C03657=1186.504,380.175,-80.249,-176.015,8.629,148.561
C03658=1186.500,380.423,-80.284,-176.014,8.633,148.561
C03659=1186.496,380.670,-80.319,-176.013,8.636,148.562
C03660=1186.492,380.918,-80.354,-176.012,8.640,148.562
C03661=1186.488,381.166,-80.388,-176.011,8.643,148.563
C03662=1186.484,381.413,-80.424,-176.010,8.646,148.564
C03663=1186.479,381.661,-80.458,-176.009,8.649,148.564
C03664=1186.476,381.908,-80.494,-176.008,8.652,148.565
C03665=1186.472,382.156,-80.528,-176.007,8.655,148.565
C03666=1186.468,382.403,-80.563,-176.006,8.658,148.566
C03667=1186.464,382.651,-80.598,-176.006,8.661,148.566
C03668=1186.460,382.898,-80.632,-176.005,8.664,148.567
C03669=1186.456,383.146,-80.668,-176.004,8.667,148.567
C03670=1186.452,383.394,-80.703,-176.003,8.671,148.568
C03671=1186.448,383.641,-80.738,-176.002,8.674,148.569
C03672=1186.444,383.889,-80.773,-176.002,8.676,148.569
C03673=1186.439,384.136,-80.808,-176.001,8.680,148.570
C03674=1186.436,384.384,-80.843,-176.000,8.683,148.570
C03675=1186.432,384.631,-80.878,-175.999,8.686,148.571
C03676=1186.428,384.878,-80.912,-175.998,8.689,148.572
C03677=1186.424,385.126,-80.948,-175.998,8.692,148.572
C03678=1186.421,385.373,-80.983,-175.997,8.695,148.573
C03679=1186.416,385.621,-81.018,-175.996,8.698,148.573
C03680=1186.412,385.868,-81.053,-175.995,8.701,148.574
C03681=1186.408,386.116,-81.088,-175.994,8.704,148.574
C03682=1186.404,386.363,-81.123,-175.995,8.707,148.575
C03683=1186.400,386.611,-81.158,-175.994,8.710,148.576
C03684=1186.396,386.858,-81.193,-175.993,8.713,148.576
C03685=1186.392,387.106,-81.229,-175.992,8.716,148.577
C03686=1186.388,387.354,-81.264,-175.991,8.719,148.577
C03687=1186.384,387.600,-81.299,-175.991,8.722,148.578
C03688=1186.380,387.848,-81.335,-175.990,8.725,148.579
C03689=1186.376,388.096,-81.369,-175.990,8.728,148.579
C03690=1186.372,388.343,-81.405,-175.990,8.730,148.580
C03691=1186.368,388.591,-81.439,-175.989,8.733,148.580
C03692=1186.365,388.839,-81.475,-175.988,8.736,148.581
C03693=1186.360,389.085,-81.510,-175.988,8.739,148.582
C03694=1186.356,389.333,-81.545,-175.987,8.742,148.582
C03695=1186.353,389.581,-81.580,-175.987,8.745,148.583
C03696=1186.348,389.828,-81.616,-175.986,8.747,148.583
C03697=1186.344,390.076,-81.651,-175.985,8.751,148.584
C03698=1186.341,390.323,-81.686,-175.986,8.753,148.585
C03699=1186.337,390.570,-81.721,-175.985,8.756,148.585
C03700=1186.333,390.818,-81.757,-175.984,8.759,148.586
C03701=1186.329,391.066,-81.792,-175.984,8.762,148.587
C03702=1186.325,391.313,-81.827,-175.983,8.765,148.587
C03703=1186.321,391.560,-81.862,-175.983,8.767,148.588
C03704=1186.316,391.844,-81.902,-175.983,8.771,148.589
C03705=1186.312,392.127,-81.943,-175.982,8.774,148.589
C03706=1186.307,392.411,-81.983,-175.982,8.777,148.590
C03707=1186.303,392.695,-82.024,-175.982,8.780,148.591
C03708=1186.298,392.943,-82.060,-175.981,8.783,148.591
C03709=1186.294,393.191,-82.095,-175.981,8.785,148.592
C03710=1186.290,393.438,-82.130,-175.980,8.788,148.593
C03711=1186.286,393.685,-82.166,-175.980,8.791,148.593
C03712=1186.283,393.933,-82.201,-175.980,8.793,148.594
C03713=1186.279,394.181,-82.236,-175.980,8.796,148.594
C03714=1186.274,394.427,-82.271,-175.979,8.799,148.595
C03715=1186.271,394.675,-82.307,-175.979,8.801,148.595
C03716=1186.267,394.922,-82.342,-175.979,8.804,148.596
C03717=1186.263,395.169,-82.378,-175.978,8.807,148.597
C03718=1186.259,395.417,-82.412,-175.978,8.809,148.597
C03719=1186.255,395.665,-82.449,-175.978,8.812,148.598
C03720=1186.251,395.913,-82.484,-175.978,8.815,148.599
C03721=1186.247,396.160,-82.519,-175.977,8.817,148.599
C03722=1186.243,396.407,-82.555,-175.977,8.819,148.600
C03723=1186.239,396.655,-82.590,-175.977,8.822,148.600
C03724=1186.235,396.902,-82.625,-175.976,8.825,148.601
C03725=1186.231,397.149,-82.660,-175.977,8.827,148.602
C03726=1186.227,397.397,-82.697,-175.976,8.830,148.602
C03727=1186.223,397.645,-82.732,-175.975,8.833,148.603
C03728=1186.219,397.892,-82.767,-175.976,8.835,148.604
C03729=1186.215,398.139,-82.803,-175.975,8.838,148.604
C03730=1186.211,398.387,-82.838,-175.975,8.840,148.605
C03731=1186.208,398.634,-82.874,-175.975,8.842,148.605
C03732=1186.203,398.881,-82.908,-175.975,8.845,148.606
C03733=1186.199,399.129,-82.945,-175.975,8.847,148.607
C03734=1186.195,399.377,-82.980,-175.974,8.850,148.607
C03735=1186.191,399.624,-83.016,-175.974,8.853,148.608
C03736=1186.187,399.871,-83.051,-175.974,8.855,148.608
C03737=1186.184,400.119,-83.086,-175.974,8.857,148.609
C03738=1186.179,400.366,-83.122,-175.974,8.860,148.609
C03739=1186.175,400.614,-83.158,-175.974,8.862,148.610
C03740=1186.171,400.861,-83.193,-175.974,8.864,148.611
C03741=1186.168,401.108,-83.229,-175.974,8.867,148.611
C03742=1186.164,401.356,-83.264,-175.974,8.869,148.612
C03743=1186.160,401.603,-83.300,-175.974,8.872,148.612
C03744=1186.156,401.851,-83.336,-175.973,8.874,148.613
C03745=1186.152,402.098,-83.371,-175.973,8.876,148.614
C03746=1186.148,402.346,-83.406,-175.973,8.879,148.614
C03747=1186.144,402.593,-83.442,-175.973,8.881,148.615
C03748=1186.140,402.841,-83.477,-175.973,8.883,148.615
C03749=1186.135,403.088,-83.513,-175.973,8.886,148.616
C03750=1186.132,403.336,-83.548,-175.973,8.888,148.616
C03751=1186.128,403.583,-83.584,-175.973,8.891,148.617
C03752=1186.124,403.831,-83.620,-175.973,8.893,148.618
C03753=1186.120,404.078,-83.656,-175.972,8.895,148.618
C03754=1186.116,404.325,-83.691,-175.972,8.897,148.619
C03755=1186.112,404.573,-83.726,-175.973,8.899,148.619
C03756=1186.108,404.820,-83.762,-175.973,8.901,148.620
C03757=1186.105,405.068,-83.798,-175.972,8.904,148.620
C03758=1186.100,405.315,-83.833,-175.972,8.906,148.621
C03759=1186.096,405.562,-83.869,-175.972,8.908,148.622
C03760=1186.092,405.810,-83.904,-175.972,8.911,148.622
C03761=1186.089,406.057,-83.940,-175.972,8.913,148.623
C03762=1186.085,406.304,-83.977,-175.972,8.916,148.623
C03763=1186.080,406.551,-84.012,-175.972,8.917,148.624
C03764=1186.077,406.799,-84.048,-175.972,8.919,148.624
C03765=1186.073,407.046,-84.083,-175.972,8.922,148.625
C03766=1186.069,407.294,-84.119,-175.972,8.924,148.626
C03767=1186.065,407.542,-84.155,-175.972,8.926,148.626
C03768=1186.061,407.789,-84.190,-175.972,8.928,148.627
C03769=1186.057,408.036,-84.225,-175.972,8.930,148.627
C03770=1186.053,408.284,-84.262,-175.972,8.933,148.628
C03771=1186.049,408.531,-84.297,-175.972,8.935,148.628
C03772=1186.045,408.779,-84.333,-175.971,8.937,148.629
C03773=1186.041,409.026,-84.369,-175.972,8.939,148.629
C03774=1186.037,409.273,-84.404,-175.972,8.941,148.630
C03775=1186.033,409.521,-84.440,-175.972,8.943,148.631
C03776=1186.029,409.768,-84.475,-175.971,8.946,148.631
C03777=1186.025,410.015,-84.512,-175.972,8.947,148.632
C03778=1186.021,410.263,-84.548,-175.971,8.949,148.632
C03779=1186.018,410.510,-84.583,-175.971,8.952,148.633
C03780=1186.014,410.757,-84.618,-175.971,8.954,148.633
C03781=1186.009,411.005,-84.654,-175.972,8.956,148.634
C03782=1186.005,411.253,-84.690,-175.971,8.958,148.634
C03783=1186.002,411.500,-84.726,-175.971,8.960,148.635
C03784=1185.997,411.748,-84.762,-175.971,8.962,148.635
C03785=1185.993,411.995,-84.797,-175.971,8.964,148.636
C03786=1185.990,412.242,-84.833,-175.971,8.966,148.637
C03787=1185.985,412.489,-84.869,-175.972,8.968,148.637
C03788=1185.982,412.737,-84.905,-175.971,8.970,148.638
C03789=1185.978,412.984,-84.940,-175.971,8.972,148.638
C03790=1185.974,413.232,-84.976,-175.971,8.974,148.639
C03791=1185.970,413.480,-85.012,-175.971,8.976,148.639
C03792=1185.966,413.726,-85.047,-175.971,8.978,148.640
C03793=1185.962,413.973,-85.083,-175.972,8.980,148.640
C03794=1185.958,414.221,-85.120,-175.971,8.982,148.641
C03795=1185.954,414.469,-85.155,-175.971,8.985,148.641
C03796=1185.951,414.716,-85.191,-175.971,8.986,148.642
C03797=1185.946,414.964,-85.227,-175.971,8.988,148.642
C03798=1185.942,415.211,-85.262,-175.971,8.990,148.643
C03799=1185.939,415.458,-85.298,-175.971,8.992,148.643
C03800=1185.932,415.876,-85.359,-175.971,8.996,148.644
C03801=1185.928,416.294,-85.419,-175.971,8.998,148.645
C03802=1185.928,416.711,-85.479,-175.971,9.002,148.646
C03803=1185.931,417.128,-85.538,-175.971,9.005,148.647
C03804=1185.510,417.129,-85.580,-175.974,9.016,148.650
C03805=1185.507,416.919,-85.550,-175.974,9.014,148.650
C03806=1185.506,416.709,-85.520,-175.974,9.012,148.649
C03807=1185.506,416.499,-85.490,-175.974,9.011,148.649
C03808=1185.506,416.289,-85.460,-175.974,9.009,148.649
C03809=1185.508,416.078,-85.429,-175.974,9.008,148.648
C03810=1185.510,415.868,-85.399,-175.974,9.006,148.648
C03811=1185.513,415.657,-85.368,-175.974,9.004,148.647
C03812=1185.517,415.448,-85.338,-175.974,9.003,148.647
C03813=1185.521,415.200,-85.302,-175.974,9.001,148.647
C03814=1185.525,414.952,-85.266,-175.974,8.999,148.646
C03815=1185.529,414.705,-85.231,-175.974,8.997,148.645
C03816=1185.533,414.457,-85.195,-175.974,8.995,148.645
C03817=1185.537,414.210,-85.158,-175.974,8.993,148.644
C03818=1185.540,413.963,-85.123,-175.975,8.991,148.644
C03819=1185.545,413.716,-85.088,-175.974,8.989,148.644
C03820=1185.549,413.468,-85.051,-175.975,8.987,148.643
C03821=1185.553,413.221,-85.016,-175.974,8.985,148.642
C03822=1185.556,412.973,-84.980,-175.974,8.983,148.642
C03823=1185.560,412.726,-84.944,-175.974,8.981,148.641
C03824=1185.564,412.478,-84.908,-175.974,8.979,148.641
C03825=1185.568,412.232,-84.873,-175.974,8.977,148.640
C03826=1185.573,411.984,-84.837,-175.975,8.975,148.640
C03827=1185.576,411.736,-84.801,-175.974,8.973,148.639
C03828=1185.580,411.489,-84.766,-175.974,8.971,148.639
C03829=1185.584,411.241,-84.730,-175.974,8.969,148.638
C03830=1185.588,410.993,-84.694,-175.975,8.966,148.638
C03831=1185.592,410.747,-84.658,-175.974,8.965,148.637
C03832=1185.596,410.500,-84.622,-175.975,8.963,148.637
C03833=1185.600,410.252,-84.586,-175.974,8.960,148.636
C03834=1185.604,410.004,-84.551,-175.974,8.959,148.635
C03835=1185.608,409.757,-84.515,-175.974,8.956,148.635
C03836=1185.611,409.509,-84.480,-175.975,8.954,148.634
C03837=1185.616,409.262,-84.444,-175.975,8.952,148.634
C03838=1185.620,409.015,-84.408,-175.974,8.950,148.633
C03839=1185.623,408.767,-84.373,-175.974,8.948,148.633
C03840=1185.628,408.520,-84.336,-175.975,8.946,148.632
C03841=1185.631,408.273,-84.300,-175.975,8.943,148.632
C03842=1185.635,408.025,-84.265,-175.974,8.942,148.631
C03843=1185.639,407.778,-84.230,-175.974,8.939,148.630
C03844=1185.644,407.531,-84.193,-175.975,8.937,148.630
C03845=1185.647,407.283,-84.158,-175.975,8.935,148.629
C03846=1185.651,407.036,-84.122,-175.975,8.932,148.629
C03847=1185.655,406.788,-84.087,-175.974,8.931,148.628
C03848=1185.660,406.541,-84.051,-175.975,8.929,148.628
C03849=1185.663,406.293,-84.016,-175.975,8.926,148.627
C03850=1185.667,406.046,-83.980,-175.975,8.924,148.626
C03851=1185.671,405.798,-83.944,-175.975,8.921,148.626
C03852=1185.675,405.551,-83.908,-175.975,8.919,148.625
C03853=1185.679,405.304,-83.873,-175.974,8.917,148.625
C03854=1185.683,405.056,-83.838,-175.975,8.915,148.624
C03855=1185.687,404.809,-83.802,-175.975,8.913,148.624
C03856=1185.691,404.561,-83.766,-175.975,8.911,148.623
C03857=1185.695,404.314,-83.730,-175.975,8.908,148.622
C03858=1185.699,404.067,-83.695,-175.975,8.906,148.622
C03859=1185.703,403.819,-83.660,-175.976,8.904,148.621
C03860=1185.707,403.571,-83.623,-175.975,8.901,148.621
C03861=1185.711,403.324,-83.588,-175.976,8.899,148.620
C03862=1185.714,403.076,-83.552,-175.976,8.896,148.620
C03863=1185.719,402.830,-83.517,-175.976,8.894,148.619
C03864=1185.722,402.582,-83.482,-175.976,8.892,148.618
C03865=1185.727,402.334,-83.445,-175.976,8.889,148.618
C03866=1185.730,402.087,-83.410,-175.976,8.887,148.617
C03867=1185.735,401.840,-83.375,-175.976,8.885,148.617
C03868=1185.738,401.593,-83.339,-175.976,8.883,148.616
C03869=1185.743,401.345,-83.303,-175.976,8.880,148.615
C03870=1185.746,401.097,-83.268,-175.977,8.877,148.615
C03871=1185.750,400.850,-83.232,-175.977,8.875,148.614
C03872=1185.754,400.603,-83.197,-175.977,8.873,148.614
C03873=1185.758,400.355,-83.161,-175.977,8.870,148.613
C03874=1185.761,400.108,-83.126,-175.977,8.868,148.612
C03875=1185.766,399.860,-83.090,-175.977,8.865,148.612
C03876=1185.770,399.613,-83.054,-175.977,8.863,148.611
C03877=1185.774,399.366,-83.019,-175.977,8.861,148.611
C03878=1185.777,399.118,-82.983,-175.977,8.858,148.610
C03879=1185.781,398.871,-82.948,-175.978,8.856,148.610
C03880=1185.786,398.623,-82.913,-175.977,8.854,148.609
C03881=1185.790,398.376,-82.877,-175.978,8.851,148.608
C03882=1185.794,398.128,-82.842,-175.979,8.848,148.608
C03883=1185.797,397.881,-82.806,-175.978,8.846,148.607
C03884=1185.802,397.634,-82.771,-175.979,8.843,148.606
C03885=1185.805,397.386,-82.735,-175.978,8.841,148.606
C03886=1185.809,397.139,-82.700,-175.979,8.839,148.605
C03887=1185.813,396.891,-82.664,-175.979,8.836,148.605
C03888=1185.818,396.644,-82.629,-175.979,8.833,148.604
C03889=1185.822,396.396,-82.594,-175.980,8.831,148.603
C03890=1185.825,396.149,-82.558,-175.980,8.828,148.603
C03891=1185.830,395.902,-82.523,-175.980,8.826,148.602
C03892=1185.833,395.654,-82.487,-175.980,8.823,148.602
C03893=1185.837,395.407,-82.452,-175.981,8.820,148.601
C03894=1185.841,395.159,-82.416,-175.980,8.818,148.600
C03895=1185.846,394.912,-82.381,-175.981,8.815,148.600
C03896=1185.850,394.664,-82.346,-175.981,8.812,148.599
C03897=1185.853,394.417,-82.310,-175.981,8.810,148.598
C03898=1185.857,394.169,-82.275,-175.982,8.807,148.598
C03899=1185.861,393.922,-82.239,-175.982,8.804,148.597
C03900=1185.865,393.674,-82.204,-175.982,8.802,148.597
C03901=1185.869,393.427,-82.169,-175.983,8.799,148.596
C03902=1185.873,393.180,-82.134,-175.983,8.796,148.595
C03903=1185.877,392.932,-82.098,-175.983,8.794,148.595
C03904=1185.881,392.684,-82.062,-175.984,8.791,148.594
C03905=1185.886,392.400,-82.022,-175.984,8.788,148.593
C03906=1185.890,392.117,-81.981,-175.985,8.784,148.593
C03907=1185.895,391.833,-81.941,-175.985,8.782,148.592
C03908=1185.899,391.550,-81.900,-175.985,8.778,148.591
C03909=1185.903,391.302,-81.866,-175.986,8.775,148.591
C03910=1185.907,391.054,-81.830,-175.986,8.773,148.590
C03911=1185.911,390.807,-81.795,-175.987,8.770,148.589
C03912=1185.915,390.560,-81.759,-175.987,8.767,148.589
C03913=1185.919,390.312,-81.724,-175.988,8.764,148.588
C03914=1185.923,390.065,-81.689,-175.988,8.762,148.588
C03915=1185.927,389.817,-81.654,-175.988,8.759,148.587
C03916=1185.931,389.569,-81.619,-175.989,8.756,148.586
C03917=1185.935,389.322,-81.584,-175.989,8.753,148.586
C03918=1185.939,389.075,-81.548,-175.990,8.750,148.585
C03919=1185.943,388.827,-81.513,-175.991,8.747,148.585
C03920=1185.947,388.580,-81.478,-175.991,8.745,148.584
C03921=1185.951,388.333,-81.443,-175.992,8.741,148.583
C03922=1185.955,388.084,-81.408,-175.992,8.738,148.583
C03923=1185.959,387.838,-81.373,-175.992,8.736,148.582
C03924=1185.963,387.590,-81.337,-175.993,8.733,148.582
C03925=1185.966,387.342,-81.302,-175.994,8.730,148.581
C03926=1185.971,387.095,-81.267,-175.994,8.727,148.580
C03927=1185.974,386.848,-81.231,-175.995,8.724,148.580
C03928=1185.978,386.600,-81.197,-175.995,8.721,148.579
C03929=1185.983,386.353,-81.161,-175.996,8.718,148.578
C03930=1185.987,386.105,-81.127,-175.997,8.715,148.578
C03931=1185.990,385.857,-81.091,-175.998,8.712,148.577
C03932=1185.995,385.610,-81.056,-175.998,8.709,148.577
C03933=1185.999,385.362,-81.021,-175.999,8.706,148.576
C03934=1186.003,385.115,-80.986,-176.000,8.703,148.576
C03935=1186.007,384.867,-80.951,-176.001,8.700,148.575
C03936=1186.010,384.620,-80.915,-176.001,8.697,148.574
C03937=1186.015,384.372,-80.881,-176.002,8.694,148.574
C03938=1186.019,384.125,-80.845,-176.002,8.690,148.573
C03939=1186.023,383.877,-80.811,-176.003,8.687,148.573
C03940=1186.027,383.630,-80.775,-176.004,8.684,148.572
C03941=1186.030,383.382,-80.741,-176.005,8.681,148.571
C03942=1186.034,383.135,-80.706,-176.006,8.678,148.571
C03943=1186.038,382.887,-80.671,-176.007,8.675,148.570
C03944=1186.042,382.640,-80.636,-176.008,8.672,148.570
C03945=1186.047,382.392,-80.601,-176.009,8.669,148.569
C03946=1186.050,382.145,-80.566,-176.009,8.666,148.569
C03947=1186.055,381.897,-80.531,-176.010,8.663,148.568
C03948=1186.058,381.650,-80.496,-176.011,8.660,148.567
C03949=1186.062,381.402,-80.461,-176.012,8.657,148.567
C03950=1186.066,381.155,-80.426,-176.013,8.653,148.566
C03951=1186.070,380.907,-80.391,-176.014,8.650,148.566
C03952=1186.074,380.660,-80.357,-176.015,8.647,148.565
C03953=1186.078,380.412,-80.321,-176.016,8.644,148.565
C03954=1186.083,380.165,-80.287,-176.017,8.641,148.564
C03955=1186.086,379.917,-80.251,-176.018,8.638,148.564
C03956=1186.090,379.669,-80.217,-176.019,8.634,148.563
C03957=1186.094,379.422,-80.183,-176.020,8.631,148.562
C03958=1186.098,379.175,-80.147,-176.021,8.628,148.562
C03959=1186.102,378.927,-80.113,-176.022,8.625,148.561
C03960=1186.106,378.679,-80.078,-176.023,8.621,148.561
C03961=1186.111,378.432,-80.043,-176.024,8.618,148.560
C03962=1186.115,378.184,-80.008,-176.025,8.615,148.560
C03963=1186.118,377.937,-79.974,-176.027,8.611,148.559
C03964=1186.122,377.690,-79.938,-176.028,8.608,148.559
C03965=1186.127,377.442,-79.904,-176.029,8.605,148.558
C03966=1186.131,377.194,-79.869,-176.030,8.601,148.557
C03967=1186.135,376.947,-79.835,-176.031,8.598,148.557
C03968=1186.138,376.699,-79.800,-176.032,8.595,148.557
C03969=1186.143,376.452,-79.765,-176.034,8.591,148.556
C03970=1186.147,376.204,-79.730,-176.035,8.588,148.556
C03971=1186.151,375.956,-79.696,-176.036,8.585,148.555
C03972=1186.154,375.709,-79.661,-176.037,8.581,148.554
C03973=1186.158,375.461,-79.626,-176.038,8.579,148.554
C03974=1186.163,375.214,-79.592,-176.040,8.575,148.553
C03975=1186.166,374.966,-79.557,-176.041,8.572,148.553
C03976=1186.170,374.719,-79.522,-176.042,8.568,148.552
C03977=1186.174,374.471,-79.487,-176.043,8.565,148.552
C03978=1186.179,374.224,-79.453,-176.045,8.561,148.551
C03979=1186.183,373.976,-79.419,-176.046,8.559,148.551
C03980=1186.187,373.728,-79.384,-176.047,8.555,148.550
C03981=1186.191,373.481,-79.350,-176.049,8.552,148.550
C03982=1186.194,373.233,-79.316,-176.051,8.548,148.549
C03983=1186.199,372.986,-79.280,-176.051,8.545,148.549
C03984=1186.203,372.738,-79.245,-176.053,8.541,148.548
C03985=1186.206,372.491,-79.212,-176.054,8.539,148.548
C03986=1186.210,372.243,-79.177,-176.056,8.535,148.547
C03987=1186.215,371.996,-79.142,-176.057,8.532,148.547
C03988=1186.218,371.748,-79.108,-176.059,8.528,148.547
C03989=1186.223,371.500,-79.074,-176.060,8.524,148.546
C03990=1186.227,371.252,-79.039,-176.061,8.522,148.546
C03991=1186.231,371.005,-79.005,-176.063,8.518,148.545
C03992=1186.235,370.758,-78.970,-176.064,8.515,148.544
C03993=1186.238,370.510,-78.936,-176.066,8.511,148.544
C03994=1186.243,370.262,-78.902,-176.068,8.508,148.544
C03995=1186.247,370.014,-78.867,-176.069,8.505,148.543
C03996=1186.251,369.767,-78.833,-176.071,8.501,148.543
C03997=1186.255,369.519,-78.798,-176.072,8.497,148.542
C03998=1186.259,369.272,-78.764,-176.073,8.494,148.542
C03999=1186.263,369.025,-78.730,-176.075,8.491,148.541
C04000=1186.267,368.776,-78.695,-176.077,8.487,148.541
C04001=1186.271,368.529,-78.661,-176.078,8.484,148.541
C04002=1186.275,368.282,-78.627,-176.080,8.481,148.540
C04003=1186.279,368.034,-78.592,-176.082,8.477,148.540
C04004=1186.284,367.786,-78.559,-176.083,8.474,148.539
C04005=1186.287,367.538,-78.524,-176.085,8.471,148.539
C04006=1186.291,367.291,-78.490,-176.087,8.467,148.538
C04007=1186.295,367.044,-78.456,-176.088,8.463,148.538
C04008=1186.299,366.796,-78.421,-176.089,8.460,148.537
C04009=1186.304,366.515,-78.383,-176.092,8.456,148.537
C04010=1186.308,366.234,-78.344,-176.093,8.452,148.536
C04011=1186.313,365.951,-78.305,-176.095,8.449,148.536
C04012=1186.317,365.670,-78.266,-176.097,8.445,148.536
C04013=1186.321,365.423,-78.232,-176.099,8.441,148.535
C04014=1186.326,365.176,-78.198,-176.101,8.438,148.535
C04015=1186.329,364.928,-78.164,-176.102,8.434,148.534
C04016=1186.334,364.680,-78.130,-176.105,8.431,148.534
C04017=1186.338,364.433,-78.096,-176.106,8.428,148.534
C04018=1186.342,364.184,-78.061,-176.108,8.424,148.533
C04019=1186.346,363.937,-78.028,-176.110,8.421,148.533
C04020=1186.350,363.690,-77.994,-176.111,8.417,148.532
C04021=1186.354,363.441,-77.959,-176.113,8.414,148.532
C04022=1186.357,363.194,-77.926,-176.115,8.410,148.532
C04023=1186.362,362.946,-77.892,-176.117,8.407,148.531
C04024=1186.366,362.699,-77.858,-176.119,8.404,148.531
C04025=1186.370,362.451,-77.824,-176.120,8.400,148.530
C04026=1186.374,362.203,-77.790,-176.123,8.397,148.530
C04027=1186.378,361.956,-77.756,-176.124,8.393,148.530
C04028=1186.382,361.708,-77.723,-176.126,8.390,148.529
C04029=1186.386,361.460,-77.688,-176.128,8.386,148.529
C04030=1186.390,361.213,-77.655,-176.130,8.384,148.529
C04031=1186.394,360.965,-77.621,-176.131,8.380,148.528
C04032=1186.398,360.717,-77.586,-176.134,8.377,148.528
C04033=1186.402,360.470,-77.553,-176.136,8.373,148.528
C04034=1186.406,360.223,-77.519,-176.138,8.370,148.527
C04035=1186.410,359.974,-77.485,-176.140,8.366,148.527
C04036=1186.414,359.727,-77.451,-176.141,8.362,148.527
C04037=1186.418,359.479,-77.418,-176.144,8.359,148.526
C04038=1186.422,359.232,-77.384,-176.145,8.355,148.526
C04039=1186.426,358.983,-77.350,-176.148,8.352,148.526
C04040=1186.430,358.736,-77.316,-176.150,8.349,148.525
C04041=1186.434,358.488,-77.283,-176.151,8.346,148.525
C04042=1186.438,358.241,-77.249,-176.153,8.342,148.525
C04043=1186.443,357.993,-77.215,-176.155,8.339,148.524
C04044=1186.447,357.745,-77.182,-176.157,8.335,148.524
C04045=1186.451,357.498,-77.148,-176.159,8.332,148.524
C04046=1186.455,357.250,-77.115,-176.162,8.329,148.524
C04047=1186.460,357.002,-77.081,-176.163,8.325,148.523
C04048=1186.463,356.755,-77.047,-176.166,8.322,148.523
C04049=1186.467,356.506,-77.014,-176.167,8.318,148.522
C04050=1186.471,356.259,-76.980,-176.170,8.315,148.522
C04051=1186.475,356.012,-76.947,-176.172,8.312,148.522
C04052=1186.479,355.764,-76.914,-176.174,8.308,148.522
C04053=1186.484,355.516,-76.880,-176.176,8.305,148.521
C04054=1186.488,355.269,-76.846,-176.178,8.301,148.521
C04055=1186.491,355.020,-76.812,-176.180,8.298,148.521
C04056=1186.495,354.772,-76.779,-176.182,8.294,148.521
C04057=1186.500,354.525,-76.746,-176.185,8.291,148.520
C04058=1186.503,354.278,-76.712,-176.186,8.287,148.520
C04059=1186.508,354.030,-76.679,-176.189,8.284,148.520
C04060=1186.512,353.782,-76.645,-176.191,8.281,148.519
C04061=1186.517,353.534,-76.612,-176.193,8.277,148.519
C04062=1186.520,353.286,-76.578,-176.195,8.274,148.519
C04063=1186.524,353.039,-76.545,-176.197,8.271,148.519
C04064=1186.528,352.791,-76.512,-176.199,8.268,148.518
C04065=1186.532,352.543,-76.478,-176.201,8.264,148.518
C04066=1186.536,352.295,-76.445,-176.203,8.261,148.518
C04067=1186.540,352.048,-76.412,-176.205,8.258,148.517
C04068=1186.545,351.800,-76.379,-176.207,8.254,148.517
C04069=1186.549,351.552,-76.346,-176.210,8.251,148.517
C04070=1186.553,351.305,-76.313,-176.211,8.248,148.517
C04071=1186.557,351.057,-76.279,-176.214,8.244,148.516
C04072=1186.561,350.810,-76.246,-176.216,8.241,148.516
C04073=1186.565,350.562,-76.213,-176.218,8.238,148.516
C04074=1186.569,350.314,-76.179,-176.220,8.234,148.516
C04075=1186.573,350.066,-76.146,-176.223,8.231,148.515
C04076=1186.577,349.818,-76.113,-176.225,8.227,148.515
C04077=1186.581,349.570,-76.080,-176.227,8.224,148.515
C04078=1186.585,349.323,-76.046,-176.229,8.221,148.515
C04079=1186.589,349.075,-76.013,-176.231,8.217,148.514
C04080=1186.593,348.827,-75.980,-176.234,8.214,148.514
C04081=1186.597,348.579,-75.947,-176.235,8.212,148.514
C04082=1186.602,348.331,-75.914,-176.237,8.208,148.514
C04083=1186.606,348.083,-75.881,-176.240,8.205,148.514
C04084=1186.610,347.836,-75.848,-176.242,8.202,148.513
C04085=1186.614,347.588,-75.815,-176.244,8.198,148.513
C04086=1186.618,347.340,-75.782,-176.246,8.195,148.513
C04087=1186.623,347.092,-75.749,-176.248,8.191,148.512
C04088=1186.627,346.845,-75.716,-176.251,8.188,148.512
C04089=1186.630,346.597,-75.683,-176.253,8.185,148.512
C04090=1186.635,346.349,-75.651,-176.255,8.181,148.512
C04091=1186.639,346.101,-75.617,-176.257,8.178,148.512
C04092=1186.643,345.853,-75.584,-176.260,8.175,148.511
C04093=1186.647,345.606,-75.551,-176.262,8.171,148.511
C04094=1186.651,345.358,-75.518,-176.264,8.168,148.511
C04095=1186.656,345.110,-75.485,-176.266,8.165,148.511
C04096=1186.659,344.862,-75.453,-176.269,8.161,148.511
C04097=1186.663,344.614,-75.420,-176.270,8.159,148.510
C04098=1186.668,344.367,-75.387,-176.272,8.156,148.510
C04099=1186.672,344.119,-75.355,-176.275,8.152,148.510
C04100=1186.676,343.871,-75.321,-176.277,8.149,148.510
C04101=1186.680,343.624,-75.289,-176.280,8.146,148.510
C04102=1186.684,343.376,-75.256,-176.282,8.143,148.509
C04103=1186.688,343.128,-75.223,-176.284,8.139,148.509
C04104=1186.693,342.880,-75.190,-176.286,8.136,148.509
C04105=1186.697,342.632,-75.158,-176.289,8.133,148.509
C04106=1186.700,342.384,-75.125,-176.291,8.129,148.509
C04107=1186.705,342.136,-75.093,-176.293,8.126,148.508
C04108=1186.709,341.888,-75.059,-176.295,8.123,148.508
C04109=1186.714,341.641,-75.027,-176.298,8.119,148.508
C04110=1186.717,341.393,-74.995,-176.300,8.116,148.508
C04111=1186.722,341.146,-74.962,-176.303,8.113,148.508
C04112=1186.726,340.897,-74.929,-176.304,8.111,148.508
C04113=1186.730,340.619,-74.893,-176.307,8.106,148.507
C04114=1186.735,340.340,-74.856,-176.309,8.103,148.507
C04115=1186.740,340.061,-74.819,-176.312,8.099,148.507
C04116=1186.745,339.783,-74.782,-176.314,8.096,148.507
C04117=1186.748,339.535,-74.751,-176.317,8.093,148.507
C04118=1186.753,339.286,-74.718,-176.319,8.089,148.506
C04119=1186.757,339.039,-74.685,-176.322,8.086,148.506
C04120=1186.761,338.790,-74.653,-176.324,8.083,148.506
C04121=1186.765,338.543,-74.620,-176.326,8.079,148.506
C04122=1186.770,338.295,-74.588,-176.329,8.076,148.506
C04123=1186.773,338.048,-74.555,-176.331,8.073,148.505
C04124=1186.778,337.799,-74.523,-176.333,8.071,148.505
C04125=1186.781,337.551,-74.491,-176.335,8.067,148.505
C04126=1186.785,337.304,-74.458,-176.337,8.064,148.505
C04127=1186.789,337.056,-74.426,-176.340,8.061,148.505
C04128=1186.794,336.808,-74.394,-176.342,8.058,148.505
C04129=1186.798,336.560,-74.361,-176.345,8.054,148.504
C04130=1186.802,336.312,-74.329,-176.347,8.051,148.504
C04131=1186.807,336.064,-74.296,-176.350,8.048,148.504
C04132=1186.810,335.816,-74.264,-176.352,8.045,148.504
C04133=1186.815,335.569,-74.232,-176.354,8.041,148.504
C04134=1186.819,335.321,-74.200,-176.357,8.038,148.504
C04135=1186.823,335.072,-74.168,-176.359,8.035,148.504
C04136=1186.826,334.825,-74.135,-176.361,8.032,148.503
C04137=1186.832,334.577,-74.103,-176.363,8.029,148.503
C04138=1186.835,334.329,-74.071,-176.366,8.026,148.503
C04139=1186.840,334.081,-74.039,-176.368,8.023,148.503
C04140=1186.843,333.833,-74.007,-176.370,8.019,148.503
C04141=1186.848,333.586,-73.974,-176.373,8.016,148.503
C04142=1186.852,333.338,-73.942,-176.375,8.013,148.503
C04143=1186.856,333.090,-73.910,-176.377,8.010,148.502
C04144=1186.860,332.841,-73.878,-176.380,8.007,148.502
C04145=1186.864,332.594,-73.846,-176.382,8.003,148.502
C04146=1186.869,332.346,-73.814,-176.384,8.001,148.502
C04147=1186.872,332.098,-73.782,-176.387,7.998,148.502
C04148=1186.877,331.850,-73.750,-176.389,7.995,148.502
C04149=1186.881,331.602,-73.718,-176.392,7.992,148.502
C04150=1186.885,331.354,-73.686,-176.394,7.988,148.502
C04151=1186.890,331.107,-73.654,-176.396,7.985,148.501
C04152=1186.893,330.859,-73.622,-176.399,7.982,148.501
C04153=1186.897,330.611,-73.590,-176.401,7.979,148.501
C04154=1186.902,330.363,-73.558,-176.403,7.975,148.501
C04155=1186.906,330.115,-73.526,-176.406,7.972,148.501
C04156=1186.910,329.867,-73.494,-176.408,7.969,148.501
C04157=1186.915,329.619,-73.463,-176.410,7.967,148.501
C04158=1186.919,329.371,-73.431,-176.413,7.964,148.501
C04159=1186.922,329.123,-73.399,-176.415,7.960,148.500
C04160=1186.927,328.875,-73.367,-176.418,7.957,148.500
C04161=1186.931,328.627,-73.335,-176.420,7.954,148.500
C04162=1186.935,328.379,-73.303,-176.423,7.951,148.500
C04163=1186.940,328.131,-73.271,-176.425,7.948,148.500
C04164=1186.943,327.883,-73.239,-176.428,7.945,148.500
C04165=1186.947,327.635,-73.208,-176.430,7.941,148.500
C04166=1186.952,327.388,-73.176,-176.432,7.939,148.500
C04167=1186.956,327.139,-73.144,-176.434,7.936,148.500
C04168=1186.961,326.892,-73.113,-176.437,7.933,148.500
C04169=1186.964,326.644,-73.081,-176.439,7.929,148.499
C04170=1186.968,326.396,-73.049,-176.441,7.926,148.499
C04171=1186.972,326.148,-73.018,-176.444,7.923,148.499
C04172=1186.977,325.899,-72.986,-176.446,7.920,148.499
C04173=1186.981,325.652,-72.954,-176.449,7.917,148.499
C04174=1186.985,325.404,-72.923,-176.451,7.913,148.499
C04175=1186.989,325.157,-72.891,-176.453,7.911,148.499
C04176=1186.993,324.908,-72.860,-176.456,7.908,148.499
C04177=1186.998,324.659,-72.828,-176.458,7.905,148.499
C04178=1187.002,324.412,-72.796,-176.461,7.902,148.498
C04179=1187.006,324.163,-72.765,-176.463,7.899,148.498
C04180=1187.010,323.916,-72.733,-176.466,7.896,148.498
C04181=1187.014,323.668,-72.702,-176.468,7.892,148.498
C04182=1187.019,323.420,-72.671,-176.471,7.889,148.498
C04183=1187.022,323.172,-72.639,-176.473,7.887,148.498
C04184=1187.027,322.925,-72.608,-176.475,7.884,148.498
C04185=1187.031,322.676,-72.576,-176.478,7.880,148.498
C04186=1187.034,322.428,-72.545,-176.480,7.877,148.498
C04187=1187.040,322.180,-72.513,-176.483,7.874,148.498
C04188=1187.044,321.932,-72.481,-176.485,7.871,148.498
C04189=1187.048,321.684,-72.451,-176.488,7.868,148.497
C04190=1187.052,321.436,-72.419,-176.490,7.865,148.497
C04191=1187.056,321.188,-72.388,-176.492,7.863,148.497
C04192=1187.060,320.940,-72.356,-176.495,7.859,148.497
C04193=1187.065,320.692,-72.325,-176.497,7.856,148.497
C04194=1187.069,320.444,-72.294,-176.500,7.853,148.497
C04195=1187.073,320.196,-72.263,-176.502,7.850,148.497
C04196=1187.077,319.949,-72.231,-176.505,7.847,148.497
C04197=1187.081,319.700,-72.200,-176.507,7.844,148.497
C04198=1187.086,319.453,-72.169,-176.510,7.841,148.497
C04199=1187.090,319.204,-72.138,-176.512,7.838,148.497
C04200=1187.094,318.957,-72.106,-176.514,7.835,148.497
C04201=1187.098,318.708,-72.075,-176.517,7.832,148.497
C04202=1187.103,318.460,-72.044,-176.519,7.829,148.497
C04203=1187.106,318.212,-72.012,-176.522,7.826,148.497
C04204=1187.111,317.964,-71.982,-176.524,7.822,148.496
C04205=1187.115,317.716,-71.951,-176.527,7.819,148.496
C04206=1187.119,317.468,-71.920,-176.529,7.817,148.496
C04207=1187.123,317.220,-71.889,-176.531,7.814,148.496
C04208=1187.127,316.972,-71.858,-176.534,7.811,148.496
C04209=1187.132,316.724,-71.826,-176.537,7.808,148.496
C04210=1187.136,316.476,-71.795,-176.539,7.805,148.496
C04211=1187.140,316.228,-71.764,-176.542,7.802,148.496
C04212=1187.145,315.980,-71.734,-176.545,7.799,148.496
C04213=1187.148,315.732,-71.702,-176.546,7.796,148.496
C04214=1187.152,315.484,-71.672,-176.549,7.793,148.496
C04215=1187.157,315.236,-71.641,-176.552,7.790,148.496
C04216=1187.161,314.987,-71.610,-176.554,7.787,148.496
C04217=1187.166,314.712,-71.575,-176.557,7.784,148.496
C04218=1187.171,314.435,-71.540,-176.560,7.780,148.496
C04219=1187.175,314.158,-71.506,-176.563,7.777,148.496
C04220=1187.180,313.882,-71.472,-176.565,7.774,148.496
C04221=1187.184,313.633,-71.441,-176.568,7.771,148.496
C04222=1187.189,313.385,-71.410,-176.570,7.768,148.496
C04223=1187.193,313.137,-71.379,-176.573,7.764,148.495
C04224=1187.196,312.889,-71.349,-176.575,7.762,148.495
C04225=1187.201,312.642,-71.317,-176.577,7.759,148.495
C04226=1187.205,312.394,-71.286,-176.580,7.756,148.495
C04227=1187.209,312.145,-71.255,-176.582,7.753,148.495
C04228=1187.213,311.897,-71.225,-176.585,7.750,148.495
C04229=1187.218,311.649,-71.194,-176.588,7.747,148.495
C04230=1187.222,311.401,-71.163,-176.589,7.744,148.495
C04231=1187.226,311.153,-71.133,-176.592,7.741,148.495
C04232=1187.230,310.905,-71.102,-176.595,7.738,148.495
C04233=1187.235,310.657,-71.072,-176.598,7.735,148.495
C04234=1187.239,310.408,-71.040,-176.600,7.732,148.495
C04235=1187.243,310.161,-71.010,-176.603,7.729,148.495
C04236=1187.248,309.912,-70.980,-176.605,7.727,148.495
C04237=1187.252,309.664,-70.949,-176.607,7.724,148.495
C04238=1187.256,309.416,-70.919,-176.610,7.720,148.495
C04239=1187.260,309.168,-70.888,-176.612,7.717,148.495
C04240=1187.265,308.920,-70.857,-176.615,7.714,148.495
C04241=1187.269,308.672,-70.827,-176.618,7.711,148.495
C04242=1187.273,308.424,-70.796,-176.619,7.709,148.495
C04243=1187.277,308.176,-70.765,-176.622,7.706,148.495
C04244=1187.282,307.928,-70.736,-176.625,7.703,148.495
C04245=1187.286,307.680,-70.705,-176.628,7.700,148.495
C04246=1187.289,307.431,-70.675,-176.630,7.697,148.495
C04247=1187.294,307.183,-70.644,-176.633,7.694,148.495
C04248=1187.299,306.935,-70.613,-176.635,7.691,148.495
C04249=1187.303,306.687,-70.584,-176.637,7.688,148.495
C04250=1187.307,306.439,-70.553,-176.640,7.685,148.495
C04251=1187.311,306.191,-70.523,-176.642,7.682,148.494
C04252=1187.315,305.943,-70.492,-176.645,7.679,148.494
C04253=1187.320,305.694,-70.462,-176.647,7.677,148.495
C04254=1187.324,305.447,-70.431,-176.650,7.674,148.495
C04255=1187.328,305.199,-70.401,-176.653,7.671,148.495
C04256=1187.333,304.950,-70.371,-176.655,7.668,148.494
C04257=1187.337,304.703,-70.341,-176.658,7.665,148.494
C04258=1187.341,304.454,-70.310,-176.660,7.662,148.494
C04259=1187.345,304.206,-70.280,-176.663,7.659,148.494
C04260=1187.350,303.958,-70.250,-176.665,7.656,148.495
C04261=1187.354,303.710,-70.219,-176.668,7.653,148.495
C04262=1187.358,303.462,-70.189,-176.670,7.650,148.494
C04263=1187.362,303.214,-70.159,-176.672,7.648,148.494
C04264=1187.367,302.965,-70.129,-176.675,7.645,148.494
C04265=1187.371,302.717,-70.099,-176.678,7.642,148.494
C04266=1187.375,302.468,-70.069,-176.680,7.639,148.494
C04267=1187.379,302.221,-70.038,-176.683,7.636,148.494
C04268=1187.383,301.972,-70.009,-176.685,7.633,148.494
C04269=1187.388,301.725,-69.978,-176.688,7.630,148.494
C04270=1187.392,301.476,-69.949,-176.690,7.627,148.494
C04271=1187.397,301.228,-69.918,-176.693,7.624,148.494
C04272=1187.401,300.980,-69.889,-176.696,7.621,148.494
C04273=1187.405,300.732,-69.858,-176.698,7.619,148.494
C04274=1187.410,300.484,-69.828,-176.701,7.616,148.494
C04275=1187.414,300.236,-69.798,-176.703,7.613,148.494
C04276=1187.418,299.988,-69.769,-176.706,7.610,148.494
C04277=1187.422,299.739,-69.738,-176.708,7.607,148.494
C04278=1187.426,299.491,-69.708,-176.710,7.605,148.494
C04279=1187.430,299.243,-69.679,-176.713,7.602,148.494
C04280=1187.435,298.995,-69.648,-176.716,7.599,148.494
C04281=1187.439,298.746,-69.618,-176.719,7.596,148.494
C04282=1187.443,298.498,-69.589,-176.721,7.594,148.495
C04283=1187.448,298.250,-69.558,-176.723,7.591,148.495
C04284=1187.452,298.002,-69.529,-176.726,7.587,148.494
C04285=1187.456,297.754,-69.499,-176.728,7.584,148.494
C04286=1187.460,297.506,-69.469,-176.731,7.581,148.494
C04287=1187.465,297.257,-69.439,-176.733,7.579,148.494
C04288=1187.469,297.009,-69.410,-176.736,7.576,148.495
C04289=1187.473,296.761,-69.380,-176.739,7.573,148.495
C04290=1187.477,296.513,-69.350,-176.741,7.570,148.495
C04291=1187.482,296.265,-69.320,-176.744,7.568,148.495
C04292=1187.486,296.016,-69.291,-176.746,7.565,148.495
C04293=1187.491,295.768,-69.261,-176.749,7.562,148.495
C04294=1187.495,295.520,-69.232,-176.752,7.559,148.495
C04295=1187.499,295.272,-69.201,-176.753,7.557,148.495
C04296=1187.503,295.024,-69.172,-176.756,7.554,148.495
C04297=1187.508,294.775,-69.142,-176.759,7.551,148.495
C04298=1187.512,294.527,-69.112,-176.762,7.548,148.495
C04299=1187.516,294.279,-69.083,-176.764,7.545,148.495
C04300=1187.520,294.031,-69.054,-176.766,7.542,148.495
C04301=1187.524,293.782,-69.024,-176.769,7.539,148.495
C04302=1187.529,293.534,-68.995,-176.772,7.536,148.495
C04303=1187.533,293.287,-68.965,-176.774,7.534,148.495
C04304=1187.538,293.039,-68.935,-176.777,7.531,148.495
C04305=1187.542,292.790,-68.905,-176.779,7.528,148.495
C04306=1187.546,292.542,-68.876,-176.782,7.525,148.495
C04307=1187.551,292.294,-68.846,-176.784,7.523,148.495
C04308=1187.555,292.045,-68.817,-176.787,7.520,148.495
C04309=1187.559,291.797,-68.788,-176.790,7.517,148.495
C04310=1187.563,291.549,-68.758,-176.792,7.514,148.495
C04311=1187.567,291.301,-68.729,-176.795,7.512,148.495
C04312=1187.571,291.052,-68.699,-176.797,7.509,148.495
C04313=1187.576,290.804,-68.670,-176.800,7.506,148.495
C04314=1187.580,290.557,-68.641,-176.802,7.503,148.495
C04315=1187.585,290.308,-68.612,-176.804,7.500,148.495
C04316=1187.589,290.059,-68.582,-176.807,7.497,148.495
C04317=1187.593,289.811,-68.553,-176.810,7.494,148.495
C04318=1187.597,289.563,-68.524,-176.813,7.491,148.495
C04319=1187.602,289.315,-68.494,-176.815,7.489,148.495
C04320=1187.606,289.066,-68.465,-176.817,7.486,148.495
C04321=1187.611,288.792,-68.432,-176.820,7.483,148.495
C04322=1187.616,288.518,-68.400,-176.823,7.481,148.496
C04323=1187.621,288.243,-68.367,-176.826,7.478,148.496
C04324=1187.626,287.968,-68.336,-176.829,7.475,148.496
C04325=1187.630,287.720,-68.306,-176.831,7.472,148.496
C04326=1187.634,287.472,-68.277,-176.834,7.469,148.496
C04327=1187.638,287.223,-68.247,-176.837,7.466,148.496
C04328=1187.643,286.975,-68.219,-176.839,7.463,148.496
C04329=1187.647,286.727,-68.190,-176.842,7.460,148.496
C04330=1187.651,286.479,-68.161,-176.845,7.457,148.496
C04331=1187.655,286.231,-68.131,-176.847,7.455,148.496
C04332=1187.660,285.982,-68.103,-176.849,7.452,148.496
C04333=1187.664,285.734,-68.073,-176.852,7.449,148.496
C04334=1187.669,285.486,-68.044,-176.855,7.446,148.496
C04335=1187.673,285.237,-68.015,-176.857,7.444,148.496
C04336=1187.677,284.989,-67.986,-176.860,7.441,148.496
C04337=1187.681,284.742,-67.957,-176.862,7.438,148.496
C04338=1187.686,284.493,-67.929,-176.865,7.436,148.496
C04339=1187.690,284.244,-67.899,-176.867,7.433,148.496
C04340=1187.694,283.996,-67.870,-176.870,7.430,148.496
C04341=1187.699,283.748,-67.841,-176.873,7.427,148.496
C04342=1187.703,283.500,-67.812,-176.875,7.425,148.496
C04343=1187.707,283.251,-67.784,-176.878,7.422,148.496
C04344=1187.711,283.003,-67.754,-176.880,7.419,148.496
C04345=1187.716,282.755,-67.726,-176.882,7.417,148.497
C04346=1187.721,282.506,-67.696,-176.885,7.414,148.497
C04347=1187.724,282.258,-67.668,-176.888,7.411,148.497
C04348=1187.729,282.010,-67.639,-176.891,7.409,148.497
C04349=1187.734,281.761,-67.610,-176.893,7.406,148.497
C04350=1187.738,281.513,-67.581,-176.896,7.403,148.497
C04351=1187.742,281.265,-67.553,-176.898,7.401,148.497
C04352=1187.747,281.016,-67.525,-176.901,7.398,148.497
C04353=1187.751,280.768,-67.495,-176.904,7.395,148.497
C04354=1187.755,280.519,-67.466,-176.906,7.392,148.497
C04355=1187.759,280.272,-67.438,-176.908,7.389,148.497
C04356=1187.764,280.023,-67.409,-176.911,7.386,148.497
C04357=1187.768,279.775,-67.380,-176.913,7.384,148.497
C04358=1187.772,279.527,-67.352,-176.916,7.381,148.497
C04359=1187.777,279.278,-67.323,-176.919,7.378,148.497
C04360=1187.780,279.030,-67.294,-176.921,7.376,148.497
C04361=1187.785,278.782,-67.266,-176.924,7.373,148.498
C04362=1187.790,278.533,-67.237,-176.927,7.370,148.498
C04363=1187.794,278.286,-67.209,-176.929,7.368,148.498
C04364=1187.798,278.037,-67.180,-176.932,7.365,148.498
C04365=1187.803,277.788,-67.151,-176.934,7.362,148.498
C04366=1187.807,277.540,-67.123,-176.937,7.360,148.498
C04367=1187.811,277.292,-67.094,-176.939,7.357,148.498
C04368=1187.815,277.043,-67.066,-176.942,7.354,148.498
C04369=1187.820,276.795,-67.037,-176.944,7.352,148.498
C04370=1187.824,276.546,-67.009,-176.947,7.349,148.498
C04371=1187.829,276.299,-66.980,-176.950,7.346,148.498
C04372=1187.833,276.050,-66.951,-176.952,7.344,148.499
C04373=1187.837,275.801,-66.923,-176.955,7.341,148.499
C04374=1187.842,275.553,-66.895,-176.958,7.338,148.499
C04375=1187.846,275.305,-66.867,-176.960,7.336,148.499
C04376=1187.851,275.057,-66.838,-176.963,7.333,148.499
C04377=1187.854,274.809,-66.810,-176.965,7.330,148.499
C04378=1187.859,274.560,-66.781,-176.968,7.328,148.499
C04379=1187.863,274.312,-66.753,-176.971,7.325,148.499
C04380=1187.868,274.063,-66.724,-176.973,7.323,148.499
C04381=1187.872,273.815,-66.697,-176.975,7.320,148.499
C04382=1187.877,273.566,-66.668,-176.978,7.317,148.499
C04383=1187.881,273.318,-66.640,-176.980,7.315,148.499
C04384=1187.885,273.070,-66.612,-176.983,7.312,148.499
C04385=1187.890,272.822,-66.584,-176.986,7.309,148.500
C04386=1187.893,272.573,-66.555,-176.988,7.307,148.500
C04387=1187.899,272.325,-66.527,-176.991,7.304,148.500
C04388=1187.902,272.076,-66.499,-176.993,7.302,148.500
C04389=1187.907,271.828,-66.470,-176.996,7.299,148.500
C04390=1187.911,271.579,-66.442,-176.999,7.296,148.500
C04391=1187.916,271.332,-66.415,-177.001,7.294,148.500
C04392=1187.920,271.083,-66.386,-177.004,7.291,148.500
C04393=1187.924,270.835,-66.358,-177.007,7.288,148.500
C04394=1187.929,270.586,-66.329,-177.009,7.286,148.500
C04395=1187.933,270.338,-66.302,-177.012,7.283,148.500
C04396=1187.937,270.089,-66.273,-177.014,7.281,148.501
C04397=1187.942,269.841,-66.246,-177.017,7.278,148.501
C04398=1187.947,269.593,-66.218,-177.020,7.275,148.501
C04399=1187.950,269.344,-66.190,-177.022,7.273,148.501
C04400=1187.956,269.096,-66.161,-177.025,7.270,148.501
C04401=1187.959,268.847,-66.133,-177.027,7.268,148.501
C04402=1187.964,268.600,-66.106,-177.030,7.265,148.501
C04403=1187.968,268.350,-66.078,-177.033,7.262,148.501
C04404=1187.973,268.102,-66.050,-177.035,7.260,148.501
C04405=1187.977,267.854,-66.022,-177.038,7.257,148.501
C04406=1187.981,267.606,-65.994,-177.040,7.255,148.502
C04407=1187.986,267.357,-65.966,-177.042,7.252,148.502
C04408=1187.990,267.108,-65.938,-177.046,7.249,148.502
C04409=1187.994,266.860,-65.910,-177.048,7.247,148.502
C04410=1187.998,266.612,-65.882,-177.051,7.244,148.502
C04411=1188.004,266.363,-65.854,-177.053,7.242,148.502
C04412=1188.008,266.115,-65.827,-177.055,7.239,148.502
C04413=1188.012,265.867,-65.799,-177.059,7.236,148.502
C04414=1188.016,265.618,-65.771,-177.061,7.234,148.502
C04415=1188.021,265.370,-65.743,-177.064,7.231,148.503
C04416=1188.025,265.121,-65.715,-177.066,7.229,148.503
C04417=1188.030,264.873,-65.688,-177.069,7.226,148.503
C04418=1188.034,264.624,-65.660,-177.071,7.224,148.503
C04419=1188.038,264.376,-65.632,-177.074,7.221,148.503
C04420=1188.043,264.128,-65.605,-177.076,7.218,148.503
C04421=1188.047,263.879,-65.576,-177.079,7.216,148.503
C04422=1188.052,263.631,-65.549,-177.082,7.213,148.503
C04423=1188.056,263.383,-65.521,-177.084,7.211,148.503
C04424=1188.060,263.133,-65.494,-177.087,7.208,148.504
C04425=1188.065,262.861,-65.464,-177.090,7.205,148.504
C04426=1188.071,262.588,-65.433,-177.093,7.202,148.504
C04427=1188.075,262.315,-65.403,-177.095,7.199,148.504
C04428=1188.080,262.043,-65.373,-177.098,7.198,148.504
C04429=1188.084,261.794,-65.345,-177.101,7.195,148.504
C04430=1188.088,261.545,-65.318,-177.103,7.192,148.504
C04431=1188.093,261.298,-65.290,-177.106,7.190,148.505
C04432=1188.097,261.048,-65.262,-177.109,7.187,148.505
C04433=1188.101,260.801,-65.235,-177.111,7.185,148.505
C04434=1188.106,260.552,-65.208,-177.114,7.182,148.505
C04435=1188.110,260.304,-65.181,-177.116,7.180,148.505
C04436=1188.114,260.055,-65.152,-177.119,7.177,148.505
C04437=1188.119,259.806,-65.125,-177.121,7.175,148.505
C04438=1188.123,259.558,-65.098,-177.124,7.172,148.505
C04439=1188.128,259.310,-65.071,-177.127,7.170,148.506
C04440=1188.132,259.061,-65.043,-177.129,7.167,148.506
C04441=1188.136,258.812,-65.016,-177.131,7.165,148.506
C04442=1188.141,258.565,-64.988,-177.135,7.162,148.506
C04443=1188.145,258.316,-64.961,-177.137,7.159,148.506
C04444=1188.149,258.067,-64.934,-177.140,7.157,148.506
C04445=1188.154,257.819,-64.906,-177.142,7.154,148.506
C04446=1188.158,257.570,-64.879,-177.145,7.152,148.506
C04447=1188.163,257.322,-64.852,-177.148,7.149,148.507
C04448=1188.167,257.073,-64.824,-177.150,7.147,148.507
C04449=1188.172,256.825,-64.797,-177.153,7.144,148.507
C04450=1188.176,256.576,-64.770,-177.155,7.142,148.507
C04451=1188.181,256.328,-64.743,-177.158,7.139,148.507
C04452=1188.185,256.079,-64.715,-177.161,7.137,148.507
C04453=1188.190,255.831,-64.688,-177.163,7.134,148.507
C04454=1188.194,255.582,-64.660,-177.165,7.132,148.508
C04455=1188.198,255.334,-64.634,-177.169,7.129,148.508
C04456=1188.202,255.086,-64.607,-177.171,7.127,148.508
C04457=1188.207,254.837,-64.580,-177.173,7.124,148.508
C04458=1188.212,254.589,-64.553,-177.176,7.122,148.508
C04459=1188.216,254.340,-64.526,-177.179,7.119,148.508
C04460=1188.220,254.091,-64.498,-177.181,7.117,148.508
C04461=1188.225,253.842,-64.471,-177.184,7.115,148.509
C04462=1188.229,253.595,-64.444,-177.186,7.112,148.509
C04463=1188.233,253.346,-64.417,-177.189,7.109,148.509
C04464=1188.238,253.098,-64.390,-177.192,7.108,148.509
C04465=1188.243,252.849,-64.363,-177.194,7.105,148.509
C04466=1188.247,252.601,-64.336,-177.197,7.102,148.509
C04467=1188.251,252.352,-64.309,-177.200,7.100,148.510
C04468=1188.255,252.104,-64.282,-177.202,7.098,148.510
C04469=1188.260,251.855,-64.255,-177.205,7.095,148.510
C04470=1188.265,251.607,-64.228,-177.207,7.093,148.510
C04471=1188.269,251.358,-64.201,-177.210,7.090,148.510
C04472=1188.273,251.110,-64.174,-177.212,7.088,148.510
C04473=1188.278,250.861,-64.148,-177.215,7.085,148.510
C04474=1188.282,250.613,-64.121,-177.218,7.083,148.511
C04475=1188.287,250.364,-64.094,-177.220,7.081,148.511
C04476=1188.291,250.116,-64.067,-177.223,7.078,148.511
C04477=1188.296,249.867,-64.040,-177.225,7.076,148.511
C04478=1188.299,249.618,-64.013,-177.228,7.073,148.511
C04479=1188.304,249.370,-63.986,-177.231,7.071,148.511
C04480=1188.309,249.121,-63.959,-177.233,7.068,148.511
C04481=1188.313,248.873,-63.933,-177.236,7.066,148.512
C04482=1188.318,248.624,-63.906,-177.239,7.063,148.512
C04483=1188.322,248.375,-63.879,-177.241,7.061,148.512
C04484=1188.326,248.127,-63.853,-177.244,7.058,148.512
C04485=1188.331,247.879,-63.826,-177.246,7.056,148.512
C04486=1188.336,247.630,-63.799,-177.249,7.054,148.513
C04487=1188.340,247.381,-63.773,-177.252,7.052,148.513
C04488=1188.344,247.133,-63.746,-177.254,7.049,148.513
C04489=1188.348,246.885,-63.719,-177.257,7.047,148.513
C04490=1188.353,246.636,-63.692,-177.259,7.045,148.513
C04491=1188.358,246.387,-63.666,-177.262,7.042,148.513
C04492=1188.362,246.139,-63.640,-177.264,7.040,148.513
C04493=1188.367,245.890,-63.612,-177.268,7.037,148.514
C04494=1188.371,245.642,-63.587,-177.270,7.035,148.514
C04495=1188.375,245.393,-63.560,-177.273,7.032,148.514
C04496=1188.379,245.145,-63.533,-177.275,7.030,148.514
C04497=1188.384,244.896,-63.507,-177.277,7.028,148.514
C04498=1188.388,244.648,-63.480,-177.281,7.025,148.515
C04499=1188.393,244.399,-63.453,-177.283,7.023,148.515
C04500=1188.397,244.150,-63.428,-177.286,7.020,148.515
C04501=1188.402,243.902,-63.401,-177.288,7.018,148.515
C04502=1188.406,243.653,-63.375,-177.291,7.015,148.515
C04503=1188.411,243.405,-63.348,-177.293,7.014,148.515
C04504=1188.415,243.156,-63.322,-177.296,7.011,148.516
C04505=1188.420,242.908,-63.295,-177.299,7.009,148.516
C04506=1188.424,242.660,-63.269,-177.301,7.007,148.516
C04507=1188.429,242.411,-63.242,-177.304,7.004,148.516
C04508=1188.433,242.163,-63.216,-177.306,7.002,148.516
C04509=1188.438,241.913,-63.190,-177.309,7.000,148.517
C04510=1188.442,241.665,-63.163,-177.312,6.997,148.517
C04511=1188.447,241.416,-63.137,-177.314,6.995,148.517
C04512=1188.451,241.168,-63.110,-177.317,6.992,148.517
C04513=1188.455,240.919,-63.085,-177.319,6.990,148.517
C04514=1188.460,240.671,-63.059,-177.322,6.988,148.518
C04515=1188.464,240.423,-63.032,-177.325,6.985,148.518
C04516=1188.469,240.173,-63.006,-177.327,6.983,148.518
C04517=1188.473,239.925,-62.979,-177.330,6.980,148.518
C04518=1188.477,239.676,-62.954,-177.333,6.979,148.518
C04519=1188.482,239.427,-62.927,-177.335,6.976,148.518
C04520=1188.486,239.179,-62.901,-177.338,6.974,148.519
C04521=1188.491,238.930,-62.875,-177.340,6.972,148.519
C04522=1188.496,238.682,-62.849,-177.343,6.969,148.519
C04523=1188.500,238.434,-62.823,-177.346,6.967,148.519
C04524=1188.504,238.185,-62.797,-177.348,6.965,148.519
C04525=1188.509,237.936,-62.770,-177.351,6.962,148.520
C04526=1188.513,237.688,-62.744,-177.354,6.960,148.520
C04527=1188.517,237.439,-62.718,-177.356,6.957,148.520
C04528=1188.523,237.190,-62.692,-177.359,6.955,148.520
C04529=1188.527,236.919,-62.664,-177.362,6.952,148.520
C04530=1188.532,236.647,-62.635,-177.364,6.951,148.521
C04531=1188.536,236.376,-62.607,-177.368,6.948,148.521
C04532=1188.542,236.104,-62.578,-177.370,6.945,148.521
C04533=1188.547,235.856,-62.553,-177.373,6.943,148.521
C04534=1188.551,235.607,-62.527,-177.375,6.941,148.521
C04535=1188.555,235.359,-62.501,-177.378,6.938,148.522
C04536=1188.560,235.109,-62.474,-177.380,6.936,148.522
C04537=1188.565,234.861,-62.449,-177.383,6.934,148.522
C04538=1188.569,234.613,-62.423,-177.386,6.931,148.522
C04539=1188.573,234.364,-62.397,-177.388,6.929,148.523
C04540=1188.577,234.115,-62.372,-177.391,6.927,148.523
C04541=1188.583,233.867,-62.345,-177.394,6.925,148.523
C04542=1188.587,233.618,-62.319,-177.396,6.923,148.523
C04543=1188.591,233.370,-62.293,-177.399,6.920,148.523
C04544=1188.595,233.121,-62.268,-177.402,6.918,148.524
C04545=1188.600,232.873,-62.242,-177.404,6.916,148.524
C04546=1188.604,232.624,-62.216,-177.407,6.913,148.524
C04547=1188.609,232.375,-62.190,-177.409,6.911,148.524
C04548=1188.614,232.127,-62.165,-177.412,6.909,148.524
C04549=1188.618,231.878,-62.139,-177.415,6.906,148.525
C04550=1188.622,231.629,-62.113,-177.417,6.904,148.525
C04551=1188.627,231.380,-62.087,-177.420,6.902,148.525
C04552=1188.632,231.132,-62.062,-177.423,6.900,148.525
C04553=1188.636,230.883,-62.036,-177.425,6.898,148.526
C04554=1188.640,230.634,-62.011,-177.428,6.896,148.526
C04555=1188.645,230.386,-61.985,-177.431,6.893,148.526
C04556=1188.649,230.138,-61.959,-177.433,6.891,148.526
C04557=1188.654,229.888,-61.933,-177.436,6.889,148.526
C04558=1188.659,229.640,-61.908,-177.438,6.886,148.526
C04559=1188.663,229.392,-61.882,-177.441,6.884,148.527
C04560=1188.668,229.142,-61.857,-177.444,6.882,148.527
C04561=1188.672,228.894,-61.832,-177.446,6.880,148.527
C04562=1188.677,228.645,-61.806,-177.449,6.878,148.528
C04563=1188.681,228.396,-61.780,-177.451,6.876,148.528
C04564=1188.686,228.148,-61.755,-177.454,6.873,148.528
C04565=1188.690,227.900,-61.729,-177.457,6.871,148.528
C04566=1188.694,227.650,-61.704,-177.459,6.869,148.528
C04567=1188.699,227.402,-61.678,-177.462,6.866,148.529
C04568=1188.703,227.153,-61.653,-177.465,6.864,148.529
C04569=1188.708,226.905,-61.627,-177.467,6.862,148.529
C04570=1188.713,226.656,-61.602,-177.471,6.860,148.529
C04571=1188.717,226.407,-61.577,-177.473,6.858,148.530
C04572=1188.722,226.159,-61.551,-177.475,6.856,148.530
C04573=1188.725,225.910,-61.526,-177.478,6.854,148.530
C04574=1188.730,225.661,-61.500,-177.481,6.851,148.530
C04575=1188.735,225.413,-61.476,-177.483,6.849,148.531
C04576=1188.739,225.164,-61.450,-177.486,6.847,148.531
C04577=1188.744,224.916,-61.424,-177.489,6.844,148.531
C04578=1188.748,224.666,-61.399,-177.491,6.842,148.531
C04579=1188.753,224.418,-61.374,-177.494,6.840,148.531
C04580=1188.757,224.169,-61.348,-177.497,6.838,148.532
C04581=1188.762,223.920,-61.323,-177.499,6.836,148.532
C04582=1188.767,223.672,-61.298,-177.502,6.834,148.532
C04583=1188.770,223.423,-61.273,-177.504,6.832,148.532
C04584=1188.775,223.175,-61.248,-177.507,6.829,148.533
C04585=1188.780,222.926,-61.222,-177.510,6.827,148.533
C04586=1188.785,222.677,-61.198,-177.512,6.825,148.533
C04587=1188.789,222.428,-61.172,-177.515,6.822,148.533
C04588=1188.794,222.180,-61.147,-177.518,6.821,148.534
C04589=1188.798,221.931,-61.122,-177.520,6.819,148.534
C04590=1188.802,221.683,-61.097,-177.523,6.817,148.534
C04591=1188.807,221.434,-61.072,-177.526,6.814,148.534
C04592=1188.812,221.186,-61.046,-177.528,6.812,148.535
C04593=1188.816,220.936,-61.021,-177.531,6.810,148.535
C04594=1188.820,220.688,-60.996,-177.533,6.808,148.535
C04595=1188.825,220.439,-60.971,-177.536,6.805,148.535
C04596=1188.830,220.191,-60.946,-177.539,6.803,148.536
C04597=1188.834,219.941,-60.921,-177.541,6.802,148.536
C04598=1188.839,219.693,-60.897,-177.544,6.799,148.536
C04599=1188.843,219.444,-60.871,-177.547,6.797,148.536
C04600=1188.848,219.195,-60.846,-177.549,6.795,148.537
C04601=1188.852,218.947,-60.821,-177.552,6.793,148.537
C04602=1188.857,218.698,-60.797,-177.555,6.790,148.537
C04603=1188.861,218.449,-60.772,-177.557,6.788,148.537
C04604=1188.866,218.201,-60.746,-177.560,6.787,148.538
C04605=1188.870,217.952,-60.722,-177.562,6.784,148.538
C04606=1188.875,217.703,-60.696,-177.565,6.782,148.538
C04607=1188.880,217.455,-60.672,-177.568,6.780,148.538
C04608=1188.884,217.206,-60.647,-177.570,6.778,148.539
C04609=1188.889,216.957,-60.623,-177.573,6.776,148.539
C04610=1188.893,216.708,-60.597,-177.576,6.773,148.539
C04611=1188.897,216.460,-60.573,-177.579,6.772,148.540
C04612=1188.902,216.210,-60.548,-177.581,6.769,148.540
C04613=1188.907,215.962,-60.522,-177.584,6.768,148.540
C04614=1188.911,215.714,-60.498,-177.587,6.765,148.540
C04615=1188.916,215.464,-60.473,-177.589,6.763,148.540
C04616=1188.920,215.216,-60.449,-177.592,6.761,148.541
C04617=1188.924,214.967,-60.423,-177.594,6.759,148.541
C04618=1188.929,214.718,-60.399,-177.597,6.757,148.541
C04619=1188.934,214.470,-60.375,-177.600,6.754,148.542
C04620=1188.938,214.221,-60.350,-177.602,6.753,148.542
C04621=1188.943,213.972,-60.326,-177.605,6.751,148.542
C04622=1188.948,213.723,-60.301,-177.607,6.749,148.542
C04623=1188.951,213.475,-60.276,-177.610,6.746,148.543
C04624=1188.956,213.226,-60.251,-177.613,6.744,148.543
C04625=1188.961,212.978,-60.227,-177.616,6.742,148.543
C04626=1188.965,212.728,-60.202,-177.618,6.740,148.543
C04627=1188.970,212.480,-60.178,-177.621,6.738,148.544
C04628=1188.974,212.231,-60.153,-177.624,6.736,148.544
C04629=1188.979,211.982,-60.129,-177.626,6.734,148.544
C04630=1188.984,211.733,-60.104,-177.629,6.732,148.545
C04631=1188.988,211.485,-60.080,-177.631,6.730,148.545
C04632=1188.993,211.236,-60.055,-177.634,6.727,148.545
C04633=1188.998,210.965,-60.028,-177.637,6.726,148.546
C04634=1189.003,210.695,-60.002,-177.640,6.723,148.546
C04635=1189.008,210.424,-59.975,-177.642,6.721,148.546
C04636=1189.012,210.155,-59.948,-177.646,6.718,148.546
C04637=1189.017,209.906,-59.924,-177.648,6.716,148.547
C04638=1189.021,209.657,-59.900,-177.651,6.715,148.547
C04639=1189.026,209.408,-59.875,-177.654,6.713,148.547
C04640=1189.030,209.160,-59.851,-177.656,6.711,148.547
C04641=1189.036,208.910,-59.827,-177.659,6.708,148.548
C04642=1189.040,208.661,-59.802,-177.662,6.706,148.548
C04643=1189.044,208.413,-59.778,-177.664,6.704,148.548
C04644=1189.049,208.164,-59.753,-177.667,6.702,148.548
C04645=1189.054,207.916,-59.729,-177.669,6.700,148.549
C04646=1189.057,207.666,-59.705,-177.672,6.698,148.549
C04647=1189.062,207.418,-59.680,-177.675,6.696,148.549
C04648=1189.067,207.169,-59.656,-177.677,6.694,148.550
C04649=1189.072,206.921,-59.631,-177.680,6.692,148.550
C04650=1189.077,206.672,-59.608,-177.683,6.690,148.550
C04651=1189.080,206.422,-59.584,-177.686,6.688,148.551
C04652=1189.086,206.174,-59.559,-177.688,6.686,148.551
C04653=1189.090,205.925,-59.535,-177.691,6.684,148.551
C04654=1189.094,205.677,-59.511,-177.693,6.682,148.551
C04655=1189.100,205.428,-59.487,-177.696,6.680,148.552
C04656=1189.104,205.178,-59.462,-177.699,6.678,148.552
C04657=1189.108,204.930,-59.438,-177.701,6.675,148.552
C04658=1189.112,204.682,-59.414,-177.704,6.673,148.553
C04659=1189.118,204.432,-59.390,-177.707,6.672,148.553
C04660=1189.122,204.184,-59.366,-177.709,6.670,148.553
C04661=1189.126,203.935,-59.342,-177.712,6.668,148.554
C04662=1189.131,203.686,-59.318,-177.714,6.666,148.554
C04663=1189.136,203.437,-59.294,-177.717,6.663,148.554
C04664=1189.140,203.189,-59.270,-177.720,6.661,148.554
C04665=1189.145,202.939,-59.246,-177.723,6.660,148.555
C04666=1189.149,202.691,-59.222,-177.725,6.658,148.555
C04667=1189.153,202.442,-59.198,-177.728,6.656,148.555
C04668=1189.159,202.193,-59.174,-177.730,6.654,148.555
C04669=1189.163,201.944,-59.150,-177.733,6.651,148.556
C04670=1189.167,201.696,-59.126,-177.736,6.649,148.556
C04671=1189.172,201.447,-59.102,-177.739,6.648,148.556
C04672=1189.176,201.198,-59.078,-177.741,6.645,148.557
C04673=1189.182,200.949,-59.054,-177.744,6.644,148.557
C04674=1189.186,200.700,-59.030,-177.746,6.642,148.557
C04675=1189.190,200.451,-59.007,-177.749,6.640,148.558
C04676=1189.195,200.202,-58.982,-177.752,6.637,148.558
C04677=1189.199,199.954,-58.958,-177.755,6.636,148.558
C04678=1189.204,199.705,-58.935,-177.757,6.633,148.558
C04679=1189.208,199.457,-58.911,-177.760,6.632,148.559
C04680=1189.213,199.208,-58.888,-177.762,6.630,148.559
C04681=1189.218,198.959,-58.863,-177.765,6.628,148.559
C04682=1189.223,198.710,-58.840,-177.768,6.626,148.560
C04683=1189.228,198.461,-58.816,-177.770,6.624,148.560
C04684=1189.232,198.212,-58.792,-177.773,6.621,148.560
C04685=1189.237,197.963,-58.769,-177.776,6.620,148.561
C04686=1189.240,197.714,-58.744,-177.778,6.618,148.561
C04687=1189.245,197.465,-58.721,-177.781,6.616,148.561
C04688=1189.250,197.217,-58.697,-177.784,6.614,148.562
C04689=1189.254,196.968,-58.674,-177.786,6.612,148.562
C04690=1189.259,196.719,-58.650,-177.789,6.610,148.562
C04691=1189.263,196.470,-58.626,-177.791,6.609,148.562
C04692=1189.268,196.221,-58.603,-177.794,6.606,148.563
C04693=1189.273,195.972,-58.579,-177.797,6.604,148.563
C04694=1189.277,195.724,-58.555,-177.800,6.602,148.563
C04695=1189.282,195.475,-58.532,-177.802,6.601,148.564
C04696=1189.286,195.226,-58.509,-177.805,6.599,148.564
C04697=1189.291,194.977,-58.485,-177.807,6.597,148.564
C04698=1189.296,194.728,-58.461,-177.810,6.595,148.565
C04699=1189.300,194.479,-58.438,-177.813,6.593,148.565
C04700=1189.305,194.230,-58.414,-177.815,6.591,148.565
C04701=1189.309,193.982,-58.390,-177.818,6.589,148.566
C04702=1189.314,193.733,-58.367,-177.821,6.587,148.566
C04703=1189.319,193.484,-58.344,-177.824,6.585,148.566
C04704=1189.323,193.235,-58.320,-177.826,6.583,148.567
C04705=1189.328,192.986,-58.296,-177.829,6.581,148.567
C04706=1189.333,192.737,-58.273,-177.831,6.579,148.567
C04707=1189.337,192.488,-58.250,-177.834,6.577,148.568
C04708=1189.341,192.240,-58.227,-177.837,6.576,148.568
C04709=1189.347,191.991,-58.204,-177.839,6.574,148.568
C04710=1189.351,191.742,-58.180,-177.842,6.572,148.569
C04711=1189.356,191.494,-58.156,-177.845,6.570,148.569
C04712=1189.360,191.245,-58.133,-177.847,6.568,148.569
C04713=1189.365,190.996,-58.110,-177.849,6.566,148.569
C04714=1189.370,190.747,-58.086,-177.853,6.564,148.570
C04715=1189.374,190.498,-58.063,-177.855,6.562,148.570
C04716=1189.378,190.249,-58.040,-177.858,6.560,148.570
C04717=1189.383,190.000,-58.017,-177.861,6.558,148.571
C04718=1189.388,189.751,-57.993,-177.863,6.556,148.571
C04719=1189.392,189.502,-57.970,-177.866,6.555,148.572
C04720=1189.397,189.253,-57.947,-177.869,6.553,148.572
C04721=1189.402,189.005,-57.924,-177.871,6.551,148.572
C04722=1189.406,188.756,-57.901,-177.874,6.549,148.572
C04723=1189.411,188.507,-57.878,-177.876,6.547,148.573
C04724=1189.416,188.258,-57.854,-177.879,6.545,148.573
C04725=1189.421,188.009,-57.831,-177.882,6.544,148.573
C04726=1189.425,187.760,-57.808,-177.884,6.542,148.574
C04727=1189.429,187.511,-57.785,-177.887,6.540,148.574
C04728=1189.434,187.262,-57.761,-177.890,6.538,148.574
C04729=1189.439,187.014,-57.738,-177.892,6.536,148.575
C04730=1189.443,186.765,-57.716,-177.895,6.535,148.575
C04731=1189.448,186.516,-57.692,-177.898,6.533,148.576
C04732=1189.453,186.267,-57.669,-177.901,6.530,148.576
C04733=1189.457,186.018,-57.646,-177.903,6.528,148.576
C04734=1189.461,185.769,-57.623,-177.906,6.526,148.576
C04735=1189.467,185.520,-57.601,-177.908,6.524,148.577
C04736=1189.472,185.271,-57.577,-177.911,6.523,148.577
C04737=1189.476,185.002,-57.553,-177.914,6.521,148.577
C04738=1189.481,184.732,-57.527,-177.916,6.519,148.578
C04739=1189.486,184.463,-57.503,-177.920,6.517,148.578
C04740=1189.491,184.193,-57.478,-177.923,6.515,148.579
C04741=1189.496,183.944,-57.455,-177.925,6.513,148.579
C04742=1189.500,183.695,-57.432,-177.928,6.511,148.579
C04743=1189.505,183.446,-57.409,-177.930,6.509,148.580
C04744=1189.510,183.197,-57.386,-177.933,6.508,148.580
C04745=1189.514,182.949,-57.363,-177.936,6.506,148.580
C04746=1189.519,182.699,-57.340,-177.938,6.504,148.581
C04747=1189.523,182.450,-57.318,-177.941,6.502,148.581
C04748=1189.528,182.201,-57.294,-177.944,6.500,148.581
C04749=1189.533,181.952,-57.272,-177.946,6.499,148.582
C04750=1189.537,181.704,-57.249,-177.949,6.497,148.582
C04751=1189.542,181.455,-57.226,-177.952,6.495,148.582
C04752=1189.546,181.206,-57.203,-177.954,6.493,148.583
C04753=1189.551,180.957,-57.181,-177.957,6.491,148.583
C04754=1189.555,180.708,-57.158,-177.960,6.490,148.583
C04755=1189.560,180.459,-57.135,-177.962,6.488,148.584
C04756=1189.565,180.211,-57.113,-177.965,6.486,148.584
C04757=1189.570,179.962,-57.090,-177.968,6.484,148.585
C04758=1189.574,179.712,-57.068,-177.970,6.482,148.585
C04759=1189.579,179.463,-57.044,-177.973,6.481,148.585
C04760=1189.583,179.215,-57.022,-177.976,6.479,148.586
C04761=1189.588,178.965,-56.999,-177.978,6.477,148.586
C04762=1189.592,178.717,-56.976,-177.981,6.475,148.586
C04763=1189.598,178.468,-56.954,-177.984,6.473,148.587
C04764=1189.602,178.219,-56.931,-177.986,6.472,148.587
C04765=1189.607,177.969,-56.909,-177.989,6.470,148.587
C04766=1189.611,177.721,-56.886,-177.992,6.468,148.588
C04767=1189.616,177.472,-56.864,-177.994,6.466,148.588
C04768=1189.620,177.223,-56.841,-177.997,6.465,148.588
C04769=1189.625,176.973,-56.818,-178.000,6.463,148.589
C04770=1189.630,176.725,-56.796,-178.002,6.461,148.589
C04771=1189.634,176.476,-56.774,-178.005,6.459,148.590
C04772=1189.639,176.228,-56.751,-178.008,6.457,148.590
C04773=1189.644,175.978,-56.729,-178.010,6.456,148.590
C04774=1189.648,175.729,-56.705,-178.013,6.454,148.591
C04775=1189.653,175.481,-56.684,-178.016,6.452,148.591
C04776=1189.658,175.231,-56.662,-178.018,6.450,148.591
C04777=1189.662,174.982,-56.638,-178.021,6.448,148.592
C04778=1189.667,174.734,-56.617,-178.024,6.447,148.592
C04779=1189.672,174.485,-56.593,-178.026,6.445,148.592
C04780=1189.676,174.235,-56.571,-178.029,6.443,148.593
C04781=1189.681,173.987,-56.550,-178.032,6.441,148.593
C04782=1189.686,173.738,-56.526,-178.034,6.440,148.594
C04783=1189.691,173.489,-56.505,-178.036,6.439,148.594
C04784=1189.695,173.240,-56.482,-178.039,6.437,148.594
C04785=1189.699,172.991,-56.459,-178.042,6.435,148.595
C04786=1189.704,172.742,-56.437,-178.044,6.433,148.595
C04787=1189.709,172.493,-56.415,-178.047,6.431,148.595
C04788=1189.714,172.244,-56.392,-178.050,6.430,148.596
C04789=1189.718,171.995,-56.370,-178.052,6.428,148.596
C04790=1189.723,171.746,-56.349,-178.055,6.426,148.596
C04791=1189.727,171.497,-56.327,-178.058,6.424,148.597
C04792=1189.733,171.249,-56.304,-178.060,6.422,148.597
C04793=1189.737,170.999,-56.282,-178.063,6.421,148.598
C04794=1189.741,170.750,-56.260,-178.066,6.419,148.598
C04795=1189.746,170.501,-56.238,-178.069,6.417,148.598
C04796=1189.751,170.252,-56.215,-178.071,6.415,148.599
C04797=1189.756,170.004,-56.193,-178.074,6.414,148.599
C04798=1189.760,169.754,-56.171,-178.077,6.412,148.599
C04799=1189.765,169.506,-56.149,-178.079,6.411,148.600
C04800=1189.770,169.256,-56.126,-178.081,6.409,148.600
C04801=1189.775,169.007,-56.105,-178.084,6.407,148.601
C04802=1189.779,168.758,-56.083,-178.087,6.405,148.601
C04803=1189.784,168.509,-56.061,-178.089,6.404,148.601
C04804=1189.788,168.261,-56.038,-178.092,6.402,148.602
C04805=1189.793,168.012,-56.016,-178.095,6.400,148.602
C04806=1189.798,167.762,-55.994,-178.097,6.398,148.602
C04807=1189.802,167.514,-55.972,-178.100,6.396,148.603
C04808=1189.807,167.264,-55.950,-178.103,6.395,148.603
C04809=1189.812,167.016,-55.929,-178.105,6.393,148.603
C04810=1189.816,166.766,-55.906,-178.108,6.391,148.604
C04811=1189.821,166.517,-55.884,-178.111,6.391,148.604
C04812=1189.826,166.268,-55.862,-178.113,6.389,148.605
C04813=1189.831,166.019,-55.840,-178.116,6.387,148.605
C04814=1189.835,165.770,-55.818,-178.119,6.385,148.606
C04815=1189.840,165.521,-55.797,-178.121,6.383,148.606
C04816=1189.845,165.273,-55.775,-178.124,6.382,148.606
C04817=1189.849,165.024,-55.753,-178.127,6.380,148.607
C04818=1189.854,164.775,-55.731,-178.129,6.378,148.607
C04819=1189.858,164.526,-55.709,-178.132,6.376,148.607
C04820=1189.863,164.277,-55.688,-178.135,6.374,148.608
C04821=1189.867,164.028,-55.666,-178.137,6.374,148.608
C04822=1189.872,163.779,-55.644,-178.140,6.372,148.609
C04823=1189.877,163.530,-55.622,-178.142,6.370,148.609
C04824=1189.881,163.280,-55.601,-178.145,6.368,148.609
C04825=1189.886,163.032,-55.579,-178.148,6.367,148.610
C04826=1189.891,162.782,-55.557,-178.151,6.365,148.610
C04827=1189.896,162.533,-55.535,-178.153,6.363,148.611
C04828=1189.900,162.284,-55.513,-178.156,6.361,148.611
C04829=1189.905,162.035,-55.491,-178.159,6.360,148.611
C04830=1189.909,161.787,-55.470,-178.161,6.359,148.612
C04831=1189.914,161.537,-55.449,-178.164,6.357,148.612
C04832=1189.919,161.288,-55.427,-178.166,6.355,148.612
C04833=1189.924,161.040,-55.405,-178.169,6.353,148.613
C04834=1189.928,160.790,-55.383,-178.172,6.352,148.613
C04835=1189.933,160.542,-55.362,-178.174,6.350,148.614
C04836=1189.938,160.293,-55.341,-178.177,6.348,148.614
C04837=1189.942,160.043,-55.319,-178.180,6.347,148.615
C04838=1189.947,159.795,-55.297,-178.182,6.346,148.615
C04839=1189.952,159.545,-55.275,-178.185,6.344,148.615
C04840=1189.957,159.296,-55.254,-178.188,6.342,148.616
C04841=1189.962,159.027,-55.230,-178.190,6.340,148.616
C04842=1189.967,158.758,-55.207,-178.193,6.338,148.616
C04843=1189.972,158.489,-55.184,-178.196,6.337,148.617
C04844=1189.977,158.220,-55.161,-178.199,6.335,148.617
C04845=1189.982,157.971,-55.139,-178.201,6.334,148.618
C04846=1189.987,157.723,-55.118,-178.204,6.332,148.618
C04847=1189.991,157.473,-55.096,-178.207,6.330,148.619
C04848=1189.996,157.224,-55.075,-178.210,6.329,148.619
C04849=1190.000,156.976,-55.053,-178.213,6.327,148.619
C04850=1190.005,156.726,-55.032,-178.215,6.326,148.620
C04851=1190.010,156.477,-55.010,-178.217,6.324,148.620
C04852=1190.015,156.228,-54.989,-178.220,6.322,148.621
C04853=1190.020,155.979,-54.968,-178.223,6.320,148.621
C04854=1190.024,155.730,-54.946,-178.225,6.319,148.621
C04855=1190.028,155.481,-54.925,-178.228,6.317,148.622
C04856=1190.033,155.232,-54.904,-178.231,6.316,148.622
C04857=1190.038,154.983,-54.883,-178.233,6.315,148.623
C04858=1190.043,154.734,-54.861,-178.236,6.313,148.623
C04859=1190.048,154.484,-54.840,-178.239,6.311,148.623
C04860=1190.052,154.236,-54.819,-178.241,6.309,148.624
C04861=1190.057,153.987,-54.798,-178.244,6.307,148.624
C04862=1190.061,153.737,-54.776,-178.246,6.306,148.625
C04863=1190.067,153.488,-54.755,-178.249,6.305,148.625
C04864=1190.071,153.240,-54.734,-178.252,6.303,148.626
C04865=1190.076,152.991,-54.713,-178.255,6.301,148.626
C04866=1190.081,152.741,-54.692,-178.257,6.300,148.626
C04867=1190.085,152.492,-54.670,-178.260,6.299,148.627
C04868=1190.090,152.243,-54.649,-178.262,6.297,148.627
C04869=1190.095,151.994,-54.627,-178.265,6.295,148.628
C04870=1190.100,151.745,-54.607,-178.268,6.294,148.628
C04871=1190.104,151.497,-54.585,-178.271,6.292,148.628
C04872=1190.109,151.247,-54.564,-178.274,6.290,148.629
C04873=1190.114,150.998,-54.543,-178.276,6.289,148.629
C04874=1190.118,150.749,-54.522,-178.278,6.288,148.630
C04875=1190.123,150.500,-54.501,-178.281,6.286,148.630
C04876=1190.128,150.251,-54.480,-178.284,6.284,148.631
C04877=1190.132,150.002,-54.459,-178.287,6.283,148.631
C04878=1190.137,149.752,-54.438,-178.289,6.282,148.631
C04879=1190.142,149.503,-54.417,-178.292,6.280,148.632
C04880=1190.146,149.255,-54.396,-178.294,6.278,148.632
C04881=1190.151,149.006,-54.375,-178.297,6.276,148.633
C04882=1190.157,148.756,-54.354,-178.300,6.276,148.633
C04883=1190.161,148.507,-54.333,-178.302,6.274,148.634
C04884=1190.165,148.258,-54.311,-178.305,6.272,148.634
C04885=1190.170,148.009,-54.291,-178.308,6.270,148.634
C04886=1190.175,147.760,-54.270,-178.310,6.269,148.635
C04887=1190.180,147.511,-54.249,-178.312,6.268,148.635
C04888=1190.184,147.262,-54.229,-178.316,6.266,148.636
C04889=1190.189,147.013,-54.207,-178.318,6.264,148.636
C04890=1190.194,146.764,-54.187,-178.321,6.263,148.636
C04891=1190.199,146.515,-54.166,-178.324,6.261,148.637
C04892=1190.203,146.266,-54.145,-178.326,6.260,148.637
C04893=1190.208,146.016,-54.124,-178.329,6.259,148.638
C04894=1190.212,145.767,-54.104,-178.332,6.257,148.638
C04895=1190.217,145.518,-54.082,-178.334,6.255,148.639
C04896=1190.222,145.269,-54.061,-178.336,6.254,148.639
C04897=1190.227,145.020,-54.040,-178.339,6.252,148.639
C04898=1190.231,144.771,-54.020,-178.342,6.251,148.640
C04899=1190.236,144.522,-53.999,-178.345,6.249,148.640
C04900=1190.241,144.273,-53.979,-178.347,6.248,148.641
C04901=1190.246,144.024,-53.958,-178.350,6.246,148.641
C04902=1190.251,143.775,-53.937,-178.352,6.245,148.642
C04903=1190.256,143.525,-53.916,-178.356,6.243,148.642
C04904=1190.260,143.276,-53.896,-178.358,6.242,148.643
C04905=1190.265,143.027,-53.875,-178.360,6.240,148.643
C04906=1190.270,142.778,-53.855,-178.363,6.239,148.643
C04907=1190.275,142.529,-53.834,-178.366,6.237,148.644
C04908=1190.279,142.280,-53.813,-178.368,6.236,148.644
C04909=1190.284,142.031,-53.793,-178.371,6.235,148.645
C04910=1190.288,141.781,-53.772,-178.374,6.233,148.645
C04911=1190.293,141.532,-53.751,-178.376,6.231,148.645
C04912=1190.298,141.283,-53.730,-178.379,6.230,148.646
C04913=1190.302,141.034,-53.710,-178.382,6.229,148.646
C04914=1190.307,140.785,-53.690,-178.384,6.227,148.647
C04915=1190.312,140.536,-53.669,-178.387,6.225,148.647
C04916=1190.316,140.287,-53.648,-178.389,6.224,148.648
C04917=1190.321,140.038,-53.628,-178.392,6.223,148.648
C04918=1190.326,139.789,-53.607,-178.395,6.221,148.649
C04919=1190.331,139.540,-53.587,-178.397,6.220,148.649
C04920=1190.336,139.291,-53.566,-178.400,6.218,148.649
C04921=1190.341,139.042,-53.546,-178.403,6.217,148.650
C04922=1190.345,138.793,-53.526,-178.406,6.215,148.650
C04923=1190.351,138.543,-53.505,-178.408,6.214,148.651
C04924=1190.355,138.294,-53.485,-178.411,6.212,148.651
C04925=1190.360,138.045,-53.464,-178.414,6.211,148.652
C04926=1190.364,137.796,-53.444,-178.416,6.210,148.652
C04927=1190.369,137.547,-53.424,-178.419,6.208,148.653
C04928=1190.374,137.298,-53.403,-178.421,6.207,148.653
C04929=1190.378,137.049,-53.383,-178.424,6.205,148.654
C04930=1190.384,136.799,-53.362,-178.427,6.204,148.654
C04931=1190.388,136.550,-53.342,-178.429,6.202,148.654
C04932=1190.393,136.301,-53.322,-178.432,6.201,148.655
C04933=1190.397,136.052,-53.302,-178.435,6.200,148.655
C04934=1190.402,135.803,-53.281,-178.437,6.198,148.656
C04935=1190.407,135.554,-53.260,-178.440,6.197,148.656
C04936=1190.412,135.305,-53.241,-178.443,6.195,148.657
C04937=1190.417,135.056,-53.221,-178.445,6.194,148.657
C04938=1190.422,134.807,-53.200,-178.448,6.192,148.658
C04939=1190.426,134.557,-53.180,-178.451,6.191,148.658
C04940=1190.431,134.308,-53.160,-178.453,6.190,148.658
C04941=1190.435,134.059,-53.139,-178.456,6.188,148.659
C04942=1190.440,133.810,-53.119,-178.459,6.187,148.659
C04943=1190.445,133.560,-53.099,-178.461,6.186,148.660
C04944=1190.450,133.312,-53.079,-178.463,6.184,148.660
C04945=1190.455,133.043,-53.057,-178.467,6.182,148.661
C04946=1190.460,132.774,-53.035,-178.469,6.181,148.661
C04947=1190.465,132.506,-53.014,-178.472,6.179,148.662
C04948=1190.470,132.237,-52.992,-178.475,6.177,148.662
C04949=1190.475,131.988,-52.972,-178.478,6.177,148.663
C04950=1190.480,131.739,-52.952,-178.480,6.175,148.663
C04951=1190.485,131.490,-52.932,-178.483,6.173,148.664
C04952=1190.489,131.240,-52.912,-178.485,6.172,148.664
C04953=1190.494,130.992,-52.892,-178.488,6.171,148.665
C04954=1190.499,130.742,-52.872,-178.491,6.169,148.665
C04955=1190.504,130.493,-52.852,-178.493,6.168,148.665
C04956=1190.509,130.244,-52.832,-178.496,6.167,148.666
C04957=1190.514,129.995,-52.812,-178.499,6.165,148.666
C04958=1190.518,129.745,-52.792,-178.501,6.164,148.667
C04959=1190.523,129.496,-52.772,-178.504,6.162,148.667
C04960=1190.528,129.248,-52.752,-178.507,6.161,148.668
C04961=1190.533,128.999,-52.732,-178.509,6.160,148.668
C04962=1190.537,128.749,-52.712,-178.512,6.158,148.669
C04963=1190.542,128.500,-52.692,-178.515,6.157,148.669
C04964=1190.546,128.250,-52.672,-178.517,6.156,148.670
C04965=1190.552,128.002,-52.653,-178.520,6.154,148.670
C04966=1190.556,127.753,-52.633,-178.523,6.153,148.670
C04967=1190.561,127.503,-52.613,-178.525,6.152,148.671
C04968=1190.565,127.254,-52.592,-178.528,6.150,148.671
C04969=1190.571,127.005,-52.573,-178.531,6.148,148.672
C04970=1190.576,126.756,-52.554,-178.533,6.148,148.672
C04971=1190.580,126.507,-52.533,-178.536,6.146,148.673
C04972=1190.585,126.257,-52.514,-178.538,6.145,148.673
C04973=1190.590,126.008,-52.494,-178.541,6.144,148.674
C04974=1190.594,125.759,-52.474,-178.544,6.142,148.674
C04975=1190.599,125.510,-52.454,-178.546,6.141,148.675
C04976=1190.604,125.260,-52.435,-178.549,6.140,148.675
C04977=1190.609,125.012,-52.415,-178.552,6.138,148.676
C04978=1190.614,124.762,-52.395,-178.554,6.137,148.676
C04979=1190.618,124.513,-52.375,-178.557,6.136,148.677
C04980=1190.624,124.264,-52.356,-178.559,6.135,148.677
C04981=1190.628,124.015,-52.336,-178.562,6.133,148.678
C04982=1190.633,123.765,-52.316,-178.565,6.131,148.678
C04983=1190.638,123.516,-52.296,-178.567,6.130,148.679
C04984=1190.642,123.267,-52.278,-178.570,6.129,148.679
C04985=1190.647,123.018,-52.257,-178.573,6.127,148.680
C04986=1190.652,122.769,-52.238,-178.575,6.126,148.680
C04987=1190.657,122.520,-52.218,-178.578,6.125,148.680
C04988=1190.662,122.270,-52.199,-178.581,6.124,148.681
C04989=1190.666,122.021,-52.179,-178.583,6.122,148.681
C04990=1190.672,121.772,-52.160,-178.586,6.121,148.682
C04991=1190.675,121.523,-52.140,-178.589,6.120,148.682
C04992=1190.680,121.274,-52.120,-178.591,6.118,148.683
C04993=1190.686,121.025,-52.101,-178.593,6.117,148.683
C04994=1190.690,120.775,-52.081,-178.597,6.116,148.684
C04995=1190.695,120.526,-52.062,-178.599,6.114,148.684
C04996=1190.700,120.277,-52.042,-178.601,6.113,148.685
C04997=1190.704,120.028,-52.023,-178.605,6.112,148.685
C04998=1190.710,119.779,-52.004,-178.607,6.111,148.686
C04999=1190.714,119.529,-51.984,-178.609,6.109,148.686
C05000=1190.719,119.280,-51.965,-178.613,6.108,148.687
C05001=1190.725,119.031,-51.945,-178.615,6.107,148.687
C05002=1190.728,118.782,-51.926,-178.617,6.105,148.688
C05003=1190.734,118.533,-51.906,-178.620,6.104,148.688
C05004=1190.738,118.284,-51.887,-178.623,6.103,148.689
C05005=1190.743,118.034,-51.867,-178.625,6.101,148.689
C05006=1190.748,117.786,-51.848,-178.628,6.100,148.690
C05007=1190.752,117.536,-51.829,-178.631,6.099,148.690
C05008=1190.758,117.287,-51.809,-178.633,6.098,148.691
C05009=1190.762,117.038,-51.790,-178.636,6.096,148.691
C05010=1190.767,116.788,-51.771,-178.638,6.095,148.691
C05011=1190.772,116.539,-51.752,-178.641,6.094,148.692
C05012=1190.777,116.289,-51.732,-178.644,6.092,148.692
C05013=1190.781,116.041,-51.714,-178.646,6.091,148.693
C05014=1190.786,115.791,-51.694,-178.649,6.090,148.693
C05015=1190.792,115.542,-51.675,-178.652,6.089,148.694
C05016=1190.796,115.293,-51.655,-178.654,6.087,148.694
C05017=1190.801,115.044,-51.636,-178.657,6.087,148.695
C05018=1190.806,114.795,-51.617,-178.660,6.085,148.695
C05019=1190.811,114.546,-51.597,-178.663,6.083,148.696
C05020=1190.815,114.296,-51.579,-178.665,6.083,148.696
C05021=1190.820,114.046,-51.559,-178.668,6.081,148.697
C05022=1190.825,113.798,-51.541,-178.670,6.080,148.697
C05023=1190.829,113.548,-51.521,-178.673,6.078,148.698
C05024=1190.835,113.299,-51.502,-178.676,6.078,148.698
C05025=1190.839,113.050,-51.483,-178.678,6.076,148.699
C05026=1190.844,112.801,-51.464,-178.681,6.074,148.699
C05027=1190.849,112.551,-51.445,-178.684,6.074,148.700
C05028=1190.854,112.302,-51.426,-178.686,6.072,148.700
C05029=1190.859,112.053,-51.406,-178.688,6.071,148.701
C05030=1190.863,111.804,-51.388,-178.692,6.070,148.701
C05031=1190.869,111.555,-51.369,-178.694,6.069,148.702
C05032=1190.874,111.305,-51.349,-178.697,6.067,148.702
C05033=1190.878,111.057,-51.331,-178.699,6.067,148.703
C05034=1190.883,110.806,-51.312,-178.702,6.065,148.703
C05035=1190.888,110.558,-51.293,-178.704,6.064,148.704
C05036=1190.893,110.308,-51.273,-178.707,6.062,148.704
C05037=1190.897,110.060,-51.255,-178.710,6.062,148.705
C05038=1190.902,109.810,-51.236,-178.712,6.060,148.705
C05039=1190.907,109.561,-51.217,-178.715,6.058,148.706
C05040=1190.912,109.311,-51.197,-178.718,6.058,148.706
C05041=1190.916,109.062,-51.179,-178.720,6.056,148.707
C05042=1190.921,108.813,-51.160,-178.723,6.055,148.707
C05043=1190.926,108.564,-51.142,-178.726,6.054,148.708
C05044=1190.931,108.315,-51.122,-178.728,6.053,148.708
C05045=1190.935,108.065,-51.103,-178.731,6.051,148.709
C05046=1190.941,107.816,-51.085,-178.733,6.051,148.709
C05047=1190.945,107.567,-51.066,-178.736,6.049,148.710
C05048=1190.951,107.317,-51.047,-178.738,6.048,148.710
C05049=1190.956,107.050,-51.027,-178.742,6.047,148.711
C05050=1190.961,106.780,-51.007,-178.744,6.045,148.711
C05051=1190.966,106.512,-50.986,-178.747,6.044,148.712
C05052=1190.971,106.244,-50.966,-178.750,6.043,148.713
C05053=1190.976,105.995,-50.947,-178.753,6.041,148.713
C05054=1190.981,105.745,-50.929,-178.755,6.040,148.713
C05055=1190.985,105.496,-50.910,-178.758,6.039,148.714
C05056=1190.991,105.247,-50.891,-178.760,6.038,148.714
C05057=1190.995,104.998,-50.872,-178.763,6.037,148.715
C05058=1191.000,104.748,-50.854,-178.766,6.036,148.716
C05059=1191.005,104.499,-50.835,-178.769,6.034,148.716
C05060=1191.010,104.250,-50.817,-178.771,6.034,148.717
C05061=1191.015,104.001,-50.797,-178.774,6.032,148.717
C05062=1191.019,103.751,-50.779,-178.776,6.031,148.718
C05063=1191.025,103.503,-50.760,-178.779,6.029,148.718
C05064=1191.029,103.253,-50.742,-178.782,6.029,148.719
C05065=1191.034,103.003,-50.724,-178.784,6.027,148.719
C05066=1191.039,102.755,-50.704,-178.787,6.027,148.720
C05067=1191.044,102.505,-50.686,-178.790,6.025,148.720
C05068=1191.048,102.256,-50.667,-178.792,6.024,148.721
C05069=1191.054,102.007,-50.649,-178.795,6.023,148.721
C05070=1191.058,101.757,-50.630,-178.797,6.022,148.722
C05071=1191.063,101.508,-50.612,-178.800,6.021,148.722
C05072=1191.068,101.259,-50.594,-178.802,6.019,148.723
C05073=1191.073,101.009,-50.575,-178.805,6.019,148.723
C05074=1191.077,100.760,-50.556,-178.808,6.017,148.724
C05075=1191.082,100.511,-50.538,-178.810,6.016,148.724
C05076=1191.088,100.262,-50.519,-178.813,6.015,148.725
C05077=1191.092,100.012,-50.500,-178.816,6.014,148.725
C05078=1191.097,99.763,-50.482,-178.818,6.012,148.726
C05079=1191.102,99.514,-50.464,-178.821,6.012,148.726
C05080=1191.107,99.264,-50.446,-178.824,6.010,148.727
C05081=1191.111,99.015,-50.427,-178.826,6.009,148.727
C05082=1191.116,98.766,-50.409,-178.829,6.008,148.728
C05083=1191.121,98.517,-50.391,-178.831,6.007,148.728
C05084=1191.126,98.267,-50.373,-178.834,6.005,148.729
C05085=1191.131,98.018,-50.353,-178.836,6.005,148.729
C05086=1191.136,97.769,-50.335,-178.840,6.003,148.730
C05087=1191.141,97.520,-50.317,-178.842,6.002,148.730
C05088=1191.145,97.270,-50.299,-178.844,6.002,148.731
C05089=1191.150,97.021,-50.281,-178.847,6.000,148.732
C05090=1191.155,96.772,-50.262,-178.850,5.999,148.732
C05091=1191.160,96.523,-50.244,-178.852,5.998,148.733
C05092=1191.165,96.274,-50.226,-178.855,5.997,148.733
C05093=1191.169,96.024,-50.207,-178.858,5.995,148.734
C05094=1191.174,95.775,-50.189,-178.860,5.995,148.734
C05095=1191.179,95.525,-50.171,-178.863,5.993,148.735
C05096=1191.185,95.276,-50.153,-178.865,5.992,148.735
C05097=1191.190,95.027,-50.135,-178.868,5.992,148.736
C05098=1191.194,94.777,-50.116,-178.871,5.990,148.736
C05099=1191.199,94.528,-50.098,-178.873,5.989,148.737
C05100=1191.204,94.279,-50.080,-178.876,5.988,148.737
C05101=1191.209,94.030,-50.062,-178.879,5.987,148.738
C05102=1191.214,93.781,-50.044,-178.881,5.985,148.738
C05103=1191.218,93.532,-50.026,-178.884,5.985,148.739
C05104=1191.223,93.282,-50.008,-178.886,5.984,148.739
C05105=1191.228,93.032,-49.989,-178.889,5.982,148.740
C05106=1191.233,92.783,-49.971,-178.891,5.981,148.740
C05107=1191.238,92.534,-49.953,-178.895,5.980,148.741
C05108=1191.243,92.285,-49.935,-178.897,5.979,148.742
C05109=1191.248,92.035,-49.917,-178.900,5.978,148.742
C05110=1191.252,91.786,-49.899,-178.902,5.977,148.743
C05111=1191.257,91.536,-49.881,-178.905,5.976,148.743
C05112=1191.262,91.287,-49.863,-178.907,5.975,148.744
C05113=1191.267,91.038,-49.845,-178.910,5.974,148.744
C05114=1191.272,90.789,-49.827,-178.913,5.972,148.745
C05115=1191.277,90.540,-49.809,-178.915,5.972,148.745
C05116=1191.282,90.291,-49.791,-178.917,5.971,148.746
C05117=1191.287,90.041,-49.773,-178.921,5.969,148.746
C05118=1191.291,89.791,-49.755,-178.923,5.969,148.747
C05119=1191.296,89.542,-49.737,-178.926,5.967,148.748
C05120=1191.301,89.293,-49.719,-178.928,5.966,148.748
C05121=1191.306,89.043,-49.701,-178.931,5.965,148.749
C05122=1191.311,88.794,-49.683,-178.933,5.964,148.749
C05123=1191.316,88.545,-49.665,-178.936,5.963,148.750
C05124=1191.321,88.296,-49.647,-178.939,5.962,148.750
C05125=1191.326,88.047,-49.629,-178.941,5.961,148.751
C05126=1191.331,87.797,-49.612,-178.944,5.959,148.751
C05127=1191.336,87.548,-49.594,-178.947,5.959,148.752
C05128=1191.341,87.299,-49.576,-178.949,5.958,148.752
C05129=1191.345,87.050,-49.559,-178.952,5.957,148.753
C05130=1191.350,86.800,-49.541,-178.954,5.956,148.753
C05131=1191.354,86.550,-49.523,-178.957,5.955,148.754
C05132=1191.359,86.301,-49.505,-178.960,5.954,148.755
C05133=1191.364,86.052,-49.487,-178.962,5.953,148.755
C05134=1191.369,85.802,-49.469,-178.965,5.951,148.756
C05135=1191.374,85.553,-49.452,-178.968,5.951,148.756
C05136=1191.379,85.303,-49.434,-178.970,5.950,148.757
C05137=1191.384,85.054,-49.416,-178.973,5.948,148.757
C05138=1191.388,84.805,-49.399,-178.975,5.948,148.758
C05139=1191.394,84.556,-49.381,-178.978,5.946,148.758
C05140=1191.399,84.306,-49.363,-178.981,5.945,148.759
C05141=1191.403,84.057,-49.345,-178.983,5.945,148.759
C05142=1191.409,83.807,-49.328,-178.986,5.943,148.760
C05143=1191.414,83.558,-49.310,-178.988,5.942,148.760
C05144=1191.418,83.309,-49.293,-178.991,5.942,148.761
C05145=1191.423,83.060,-49.275,-178.994,5.940,148.761
C05146=1191.428,82.810,-49.257,-178.996,5.939,148.762
C05147=1191.433,82.561,-49.240,-178.998,5.938,148.763
C05148=1191.438,82.312,-49.222,-179.002,5.937,148.763
C05149=1191.442,82.063,-49.205,-179.004,5.937,148.764
C05150=1191.447,81.813,-49.188,-179.007,5.935,148.764
C05151=1191.452,81.564,-49.170,-179.010,5.934,148.765
C05152=1191.457,81.315,-49.152,-179.012,5.933,148.765
C05153=1191.463,81.046,-49.133,-179.015,5.932,148.766
C05154=1191.468,80.778,-49.115,-179.018,5.931,148.767
C05155=1191.473,80.510,-49.096,-179.020,5.930,148.767
C05156=1191.478,80.241,-49.077,-179.023,5.929,148.768
C05157=1191.483,79.991,-49.059,-179.026,5.928,148.768
C05158=1191.488,79.742,-49.042,-179.028,5.927,148.769
C05159=1191.493,79.493,-49.024,-179.031,5.926,148.769
C05160=1191.498,79.244,-49.008,-179.034,5.925,148.770
C05161=1191.503,78.995,-48.990,-179.036,5.924,148.771
C05162=1191.508,78.745,-48.973,-179.038,5.923,148.771
C05163=1191.513,78.496,-48.955,-179.042,5.922,148.772
C05164=1191.518,78.246,-48.938,-179.044,5.921,148.772
C05165=1191.523,77.997,-48.920,-179.046,5.920,148.773
C05166=1191.527,77.747,-48.903,-179.050,5.919,148.773
C05167=1191.532,77.498,-48.885,-179.052,5.918,148.774
C05168=1191.538,77.248,-48.868,-179.054,5.918,148.774
C05169=1191.542,77.000,-48.850,-179.057,5.916,148.775
C05170=1191.548,76.751,-48.834,-179.060,5.915,148.775
C05171=1191.553,76.501,-48.816,-179.062,5.915,148.776
C05172=1191.557,76.252,-48.799,-179.065,5.913,148.777
C05173=1191.562,76.002,-48.782,-179.068,5.912,148.777
C05174=1191.567,75.753,-48.765,-179.070,5.912,148.778
C05175=1191.572,75.503,-48.747,-179.073,5.910,148.778
C05176=1191.577,75.254,-48.730,-179.075,5.909,148.779
C05177=1191.581,75.005,-48.712,-179.078,5.909,148.779
C05178=1191.587,74.756,-48.695,-179.081,5.907,148.780
C05179=1191.591,74.506,-48.679,-179.083,5.906,148.780
C05180=1191.596,74.257,-48.661,-179.086,5.906,148.781
C05181=1191.601,74.007,-48.643,-179.088,5.904,148.782
C05182=1191.606,73.758,-48.627,-179.091,5.904,148.782
C05183=1191.611,73.508,-48.610,-179.093,5.903,148.783
C05184=1191.616,73.260,-48.593,-179.096,5.901,148.783
C05185=1191.621,73.010,-48.575,-179.099,5.901,148.784
C05186=1191.626,72.760,-48.559,-179.101,5.900,148.784
C05187=1191.631,72.511,-48.541,-179.104,5.899,148.785
C05188=1191.636,72.261,-48.523,-179.107,5.898,148.785
C05189=1191.641,72.013,-48.507,-179.109,5.897,148.786
C05190=1191.646,71.763,-48.490,-179.111,5.896,148.787
C05191=1191.650,71.513,-48.473,-179.115,5.895,148.787
C05192=1191.655,71.264,-48.455,-179.117,5.894,148.788
C05193=1191.660,71.015,-48.438,-179.119,5.893,148.788
C05194=1191.666,70.766,-48.422,-179.122,5.892,148.789
C05195=1191.670,70.516,-48.405,-179.125,5.891,148.789
C05196=1191.675,70.266,-48.388,-179.127,5.891,148.790
C05197=1191.680,70.018,-48.370,-179.130,5.890,148.791
C05198=1191.685,69.768,-48.353,-179.133,5.888,148.791
C05199=1191.690,69.519,-48.337,-179.135,5.888,148.792
C05200=1191.694,69.269,-48.320,-179.137,5.887,148.792
C05201=1191.700,69.020,-48.303,-179.141,5.886,148.793
C05202=1191.704,68.770,-48.286,-179.143,5.885,148.794
C05203=1191.710,68.521,-48.269,-179.145,5.884,148.794
C05204=1191.714,68.272,-48.253,-179.148,5.884,148.795
C05205=1191.720,68.022,-48.235,-179.151,5.882,148.795
C05206=1191.724,67.773,-48.218,-179.153,5.881,148.796
C05207=1191.729,67.524,-48.202,-179.156,5.881,148.796
C05208=1191.734,67.274,-48.184,-179.159,5.879,148.797
C05209=1191.738,67.025,-48.168,-179.161,5.879,148.797
C05210=1191.744,66.775,-48.150,-179.163,5.878,148.798
C05211=1191.749,66.526,-48.134,-179.166,5.877,148.799
C05212=1191.753,66.277,-48.117,-179.169,5.876,148.799
C05213=1191.758,66.027,-48.100,-179.171,5.875,148.800
C05214=1191.764,65.778,-48.084,-179.174,5.874,148.800
C05215=1191.769,65.528,-48.067,-179.176,5.873,148.801
C05216=1191.773,65.279,-48.050,-179.179,5.872,148.801
C05217=1191.778,65.030,-48.034,-179.182,5.872,148.802
C05218=1191.784,64.780,-48.016,-179.184,5.871,148.803
C05219=1191.788,64.531,-48.000,-179.187,5.870,148.803
C05220=1191.793,64.282,-47.983,-179.190,5.868,148.804
C05221=1191.798,64.032,-47.966,-179.192,5.868,148.804
C05222=1191.803,63.783,-47.949,-179.195,5.867,148.805
C05223=1191.807,63.533,-47.933,-179.197,5.866,148.805
C05224=1191.813,63.284,-47.917,-179.200,5.865,148.806
C05225=1191.818,63.034,-47.900,-179.203,5.865,148.807
C05226=1191.823,62.785,-47.884,-179.205,5.864,148.807
C05227=1191.827,62.536,-47.867,-179.208,5.863,148.808
C05228=1191.833,62.286,-47.850,-179.210,5.861,148.808
C05229=1191.838,62.037,-47.833,-179.213,5.861,148.809
C05230=1191.842,61.788,-47.817,-179.216,5.860,148.810
C05231=1191.847,61.538,-47.800,-179.218,5.859,148.810
C05232=1191.853,61.289,-47.784,-179.221,5.858,148.811
C05233=1191.857,61.039,-47.767,-179.224,5.858,148.811
C05234=1191.862,60.790,-47.750,-179.226,5.857,148.812
C05235=1191.867,60.541,-47.734,-179.228,5.856,148.812
C05236=1191.872,60.291,-47.717,-179.231,5.854,148.813
C05237=1191.877,60.042,-47.701,-179.234,5.854,148.814
C05238=1191.882,59.792,-47.685,-179.236,5.853,148.814
C05239=1191.886,59.543,-47.668,-179.239,5.852,148.815
C05240=1191.892,59.294,-47.651,-179.242,5.851,148.815
C05241=1191.897,59.044,-47.634,-179.244,5.851,148.816
C05242=1191.902,58.795,-47.619,-179.247,5.850,148.816
C05243=1191.907,58.545,-47.602,-179.249,5.849,148.817
C05244=1191.911,58.296,-47.586,-179.252,5.849,148.818
C05245=1191.917,58.047,-47.569,-179.255,5.847,148.818
C05246=1191.922,57.797,-47.553,-179.257,5.846,148.819
C05247=1191.927,57.548,-47.536,-179.259,5.845,148.819
C05248=1191.931,57.298,-47.520,-179.262,5.845,148.820
C05249=1191.937,57.049,-47.504,-179.265,5.844,148.821
C05250=1191.941,56.799,-47.487,-179.267,5.843,148.821
C05251=1191.946,56.551,-47.471,-179.270,5.842,148.822
C05252=1191.952,56.300,-47.455,-179.273,5.842,148.822
C05253=1191.956,56.051,-47.438,-179.275,5.841,148.823
C05254=1191.961,55.802,-47.422,-179.278,5.839,148.823
C05255=1191.966,55.552,-47.406,-179.281,5.839,148.824
C05256=1191.971,55.303,-47.389,-179.283,5.838,148.825
C05257=1191.977,55.035,-47.372,-179.285,5.837,148.825
C05258=1191.981,54.766,-47.354,-179.289,5.836,148.826
C05259=1191.988,54.497,-47.337,-179.291,5.836,148.827
C05260=1191.993,54.229,-47.319,-179.294,5.835,148.827
C05261=1191.998,53.979,-47.303,-179.297,5.833,148.828
C05262=1192.003,53.730,-47.287,-179.299,5.833,148.828
C05263=1192.008,53.480,-47.271,-179.302,5.832,148.829
C05264=1192.013,53.232,-47.254,-179.304,5.831,148.829
C05265=1192.017,52.981,-47.238,-179.307,5.831,148.830
C05266=1192.022,52.733,-47.222,-179.310,5.830,148.831
C05267=1192.027,52.483,-47.206,-179.312,5.829,148.831
C05268=1192.032,52.234,-47.190,-179.315,5.828,148.832
C05269=1192.037,51.984,-47.174,-179.317,5.828,148.833
C05270=1192.042,51.735,-47.158,-179.319,5.827,148.833
C05271=1192.047,51.485,-47.142,-179.323,5.825,148.834
C05272=1192.052,51.236,-47.125,-179.325,5.825,148.834
C05273=1192.057,50.986,-47.109,-179.327,5.824,148.835
C05274=1192.062,50.737,-47.093,-179.330,5.823,148.835
C05275=1192.067,50.487,-47.077,-179.333,5.823,148.836
C05276=1192.072,50.238,-47.061,-179.335,5.822,148.837
C05277=1192.077,49.988,-47.045,-179.338,5.821,148.837
C05278=1192.082,49.739,-47.029,-179.341,5.820,148.838
C05279=1192.087,49.490,-47.013,-179.343,5.819,148.838
C05280=1192.092,49.240,-46.997,-179.345,5.819,148.839
C05281=1192.097,48.991,-46.981,-179.348,5.818,148.840
C05282=1192.102,48.741,-46.965,-179.350,5.817,148.840
C05283=1192.107,48.492,-46.948,-179.354,5.816,148.841
C05284=1192.112,48.242,-46.933,-179.356,5.815,148.841
C05285=1192.117,47.993,-46.917,-179.358,5.815,148.842
C05286=1192.122,47.744,-46.901,-179.361,5.814,148.843
C05287=1192.126,47.494,-46.885,-179.364,5.814,148.843
C05288=1192.131,47.245,-46.870,-179.366,5.813,148.844
C05289=1192.136,46.995,-46.853,-179.369,5.811,148.844
C05290=1192.141,46.746,-46.837,-179.372,5.811,148.845
C05291=1192.147,46.496,-46.822,-179.374,5.810,148.845
C05292=1192.151,46.247,-46.805,-179.376,5.809,148.846
C05293=1192.157,45.998,-46.790,-179.379,5.809,148.847
C05294=1192.161,45.747,-46.774,-179.381,5.808,148.847
C05295=1192.166,45.499,-46.758,-179.384,5.807,148.848
C05296=1192.171,45.250,-46.742,-179.387,5.806,148.849
C05297=1192.176,44.999,-46.726,-179.389,5.805,148.849
C05298=1192.181,44.750,-46.711,-179.392,5.805,148.850
C05299=1192.186,44.501,-46.694,-179.394,5.804,148.850
C05300=1192.191,44.251,-46.679,-179.397,5.803,148.851
C05301=1192.197,44.002,-46.663,-179.399,5.803,148.851
C05302=1192.201,43.753,-46.648,-179.402,5.802,148.852
C05303=1192.206,43.503,-46.632,-179.405,5.801,148.853
C05304=1192.211,43.254,-46.616,-179.407,5.800,148.853
C05305=1192.216,43.004,-46.600,-179.410,5.800,148.854
C05306=1192.221,42.754,-46.584,-179.412,5.799,148.854
C05307=1192.226,42.505,-46.569,-179.415,5.798,148.855
C05308=1192.231,42.256,-46.554,-179.417,5.798,148.856
C05309=1192.236,42.006,-46.537,-179.420,5.797,148.856
C05310=1192.241,41.757,-46.521,-179.423,5.795,148.857
C05311=1192.247,41.508,-46.506,-179.425,5.795,148.857
C05312=1192.251,41.258,-46.490,-179.428,5.794,148.858
C05313=1192.256,41.008,-46.475,-179.430,5.793,148.859
C05314=1192.261,40.759,-46.459,-179.433,5.793,148.859
C05315=1192.267,40.510,-46.444,-179.435,5.792,148.860
C05316=1192.271,40.260,-46.428,-179.438,5.792,148.860
C05317=1192.276,40.010,-46.413,-179.440,5.791,148.861
C05318=1192.281,39.762,-46.396,-179.443,5.790,148.862
C05319=1192.285,39.512,-46.381,-179.446,5.789,148.862
C05320=1192.291,39.262,-46.365,-179.448,5.788,148.863
C05321=1192.296,39.013,-46.350,-179.451,5.788,148.864
C05322=1192.301,38.764,-46.334,-179.454,5.787,148.864
C05323=1192.306,38.514,-46.319,-179.456,5.786,148.865
C05324=1192.311,38.264,-46.303,-179.458,5.786,148.865
C05325=1192.316,38.015,-46.288,-179.461,5.785,148.866
C05326=1192.321,37.766,-46.273,-179.463,5.784,148.866
C05327=1192.326,37.516,-46.257,-179.466,5.783,148.867
C05328=1192.331,37.266,-46.241,-179.469,5.783,148.868
C05329=1192.336,37.017,-46.226,-179.472,5.782,148.868
C05330=1192.341,36.768,-46.211,-179.474,5.781,148.869
C05331=1192.346,36.518,-46.195,-179.476,5.781,148.870
C05332=1192.351,36.269,-46.180,-179.479,5.780,148.870
C05333=1192.356,36.019,-46.164,-179.481,5.779,148.871
C05334=1192.361,35.770,-46.148,-179.484,5.779,148.871
C05335=1192.366,35.521,-46.133,-179.486,5.778,148.872
C05336=1192.371,35.270,-46.118,-179.489,5.777,148.873
C05337=1192.376,35.021,-46.103,-179.491,5.777,148.873
C05338=1192.381,34.772,-46.088,-179.495,5.776,148.874
C05339=1192.387,34.522,-46.072,-179.497,5.775,148.875
C05340=1192.391,34.273,-46.057,-179.499,5.774,148.875
C05341=1192.396,34.023,-46.041,-179.502,5.774,148.876
C05342=1192.401,33.774,-46.026,-179.505,5.773,148.876
C05343=1192.406,33.524,-46.011,-179.507,5.772,148.877
C05344=1192.411,33.275,-45.996,-179.509,5.772,148.877
C05345=1192.416,33.025,-45.981,-179.512,5.771,148.878
C05346=1192.422,32.776,-45.965,-179.515,5.771,148.879
C05347=1192.426,32.526,-45.950,-179.517,5.770,148.879
C05348=1192.431,32.277,-45.934,-179.519,5.769,148.880
C05349=1192.436,32.028,-45.919,-179.522,5.769,148.881
C05350=1192.441,31.778,-45.904,-179.525,5.767,148.881
C05351=1192.446,31.529,-45.889,-179.528,5.767,148.882
C05352=1192.452,31.279,-45.874,-179.530,5.766,148.882
C05353=1192.456,31.029,-45.858,-179.533,5.766,148.883
C05354=1192.461,30.780,-45.843,-179.535,5.765,148.884
C05355=1192.466,30.530,-45.828,-179.538,5.764,148.884
C05356=1192.471,30.281,-45.813,-179.540,5.764,148.885
C05357=1192.476,30.032,-45.798,-179.543,5.763,148.886
C05358=1192.481,29.782,-45.782,-179.545,5.762,148.886
C05359=1192.486,29.533,-45.768,-179.548,5.762,148.887
C05360=1192.492,29.283,-45.752,-179.550,5.761,148.887
C05361=1192.497,29.014,-45.737,-179.553,5.761,148.888
C05362=1192.502,28.746,-45.720,-179.556,5.760,148.889
C05363=1192.507,28.477,-45.704,-179.558,5.759,148.889
C05364=1192.513,28.208,-45.688,-179.561,5.758,148.890
C05365=1192.517,27.958,-45.672,-179.564,5.758,148.891
C05366=1192.523,27.709,-45.657,-179.566,5.757,148.891
C05367=1192.528,27.459,-45.642,-179.569,5.757,148.892
C05368=1192.533,27.210,-45.627,-179.571,5.756,148.892
C05369=1192.538,26.960,-45.613,-179.574,5.755,148.893
C05370=1192.543,26.711,-45.598,-179.576,5.755,148.894
C05371=1192.548,26.462,-45.582,-179.579,5.754,148.894
C05372=1192.553,26.212,-45.568,-179.582,5.753,148.895
C05373=1192.558,25.962,-45.552,-179.584,5.752,148.896
C05374=1192.563,25.713,-45.537,-179.587,5.752,148.896
C05375=1192.568,25.464,-45.523,-179.589,5.751,148.897
C05376=1192.573,25.214,-45.507,-179.592,5.750,148.897
C05377=1192.578,24.965,-45.493,-179.595,5.750,148.898
C05378=1192.583,24.715,-45.478,-179.597,5.749,148.899
C05379=1192.589,24.465,-45.463,-179.599,5.748,148.899
C05380=1192.593,24.216,-45.448,-179.602,5.748,148.900
C05381=1192.598,23.967,-45.434,-179.605,5.747,148.900
C05382=1192.604,23.717,-45.418,-179.607,5.747,148.901
C05383=1192.608,23.467,-45.404,-179.609,5.746,148.902
C05384=1192.613,23.218,-45.389,-179.612,5.745,148.902
C05385=1192.618,22.968,-45.373,-179.615,5.745,148.903
C05386=1192.623,22.719,-45.359,-179.617,5.744,148.904
C05387=1192.628,22.469,-45.345,-179.620,5.744,148.904
C05388=1192.633,22.219,-45.329,-179.622,5.743,148.905
C05389=1192.638,21.970,-45.315,-179.625,5.743,148.905
C05390=1192.643,21.721,-45.300,-179.627,5.742,148.906
C05391=1192.649,21.471,-45.285,-179.630,5.741,148.907
C05392=1192.653,21.222,-45.270,-179.632,5.741,148.907
C05393=1192.658,20.972,-45.256,-179.635,5.740,148.908
C05394=1192.664,20.723,-45.241,-179.638,5.740,148.909
C05395=1192.669,20.473,-45.226,-179.640,5.739,148.909
C05396=1192.674,20.224,-45.212,-179.642,5.738,148.910
C05397=1192.679,19.975,-45.197,-179.645,5.738,148.910
C05398=1192.684,19.725,-45.182,-179.647,5.737,148.911
C05399=1192.689,19.476,-45.167,-179.650,5.736,148.912
C05400=1192.694,19.226,-45.153,-179.653,5.736,148.912
C05401=1192.699,18.976,-45.138,-179.655,5.735,148.913
C05402=1192.704,18.727,-45.123,-179.657,5.735,148.913
C05403=1192.709,18.477,-45.109,-179.660,5.734,148.914
C05404=1192.714,18.227,-45.094,-179.663,5.734,148.915
C05405=1192.719,17.978,-45.079,-179.665,5.733,148.915
C05406=1192.724,17.728,-45.065,-179.667,5.732,148.916
C05407=1192.729,17.479,-45.051,-179.670,5.732,148.917
C05408=1192.734,17.230,-45.036,-179.673,5.731,148.917
C05409=1192.739,16.980,-45.021,-179.675,5.731,148.918
C05410=1192.744,16.730,-45.006,-179.678,5.730,148.918
C05411=1192.749,16.481,-44.992,-179.680,5.729,148.919
C05412=1192.754,16.232,-44.978,-179.683,5.729,148.920
C05413=1192.759,15.982,-44.963,-179.685,5.728,148.920
C05414=1192.764,15.732,-44.949,-179.688,5.728,148.921
C05415=1192.770,15.483,-44.933,-179.690,5.727,148.922
C05416=1192.775,15.233,-44.919,-179.693,5.726,148.922
C05417=1192.780,14.984,-44.905,-179.696,5.726,148.923
C05418=1192.785,14.734,-44.891,-179.698,5.725,148.924
C05419=1192.789,14.485,-44.876,-179.700,5.725,148.924
C05420=1192.794,14.235,-44.861,-179.703,5.724,148.925
C05421=1192.800,13.986,-44.847,-179.706,5.724,148.925
C05422=1192.805,13.736,-44.833,-179.708,5.723,148.926
C05423=1192.810,13.487,-44.819,-179.711,5.722,148.927
C05424=1192.815,13.237,-44.804,-179.713,5.722,148.927
C05425=1192.820,12.988,-44.789,-179.716,5.721,148.928
C05426=1192.825,12.738,-44.775,-179.718,5.721,148.929
C05427=1192.830,12.488,-44.760,-179.721,5.720,148.929
C05428=1192.836,12.239,-44.747,-179.723,5.719,148.930
C05429=1192.840,11.989,-44.732,-179.726,5.719,148.930
C05430=1192.845,11.740,-44.718,-179.729,5.718,148.931
C05431=1192.850,11.490,-44.704,-179.731,5.718,148.932
C05432=1192.855,11.241,-44.689,-179.733,5.717,148.932
C05433=1192.860,10.991,-44.674,-179.736,5.717,148.933
C05434=1192.866,10.742,-44.661,-179.739,5.716,148.934
C05435=1192.871,10.492,-44.646,-179.741,5.715,148.934
C05436=1192.875,10.243,-44.632,-179.744,5.715,148.935
C05437=1192.880,9.993,-44.618,-179.746,5.714,148.936
C05438=1192.885,9.743,-44.603,-179.749,5.714,148.936
C05439=1192.891,9.494,-44.590,-179.751,5.713,148.937
C05440=1192.896,9.245,-44.575,-179.754,5.712,148.937
C05441=1192.901,8.995,-44.561,-179.756,5.712,148.938
C05442=1192.906,8.745,-44.547,-179.759,5.711,148.939
C05443=1192.911,8.495,-44.532,-179.761,5.712,148.939
C05444=1192.916,8.246,-44.519,-179.763,5.711,148.940
C05445=1192.921,7.997,-44.504,-179.766,5.710,148.941
C05446=1192.926,7.747,-44.490,-179.768,5.710,148.941
C05447=1192.931,7.497,-44.476,-179.771,5.709,148.942
C05448=1192.936,7.248,-44.461,-179.773,5.708,148.942
C05449=1192.942,6.999,-44.447,-179.776,5.708,148.943
C05450=1192.947,6.749,-44.433,-179.779,5.708,148.944
C05451=1192.952,6.499,-44.419,-179.781,5.707,148.944
C05452=1192.957,6.249,-44.405,-179.783,5.706,148.945
C05453=1192.962,6.000,-44.391,-179.786,5.706,148.946
C05454=1192.967,5.751,-44.376,-179.789,5.705,148.946
C05455=1192.971,5.501,-44.363,-179.791,5.705,148.947
C05456=1192.976,5.252,-44.349,-179.794,5.704,148.948
C05457=1192.982,5.003,-44.335,-179.796,5.703,148.948
C05458=1192.987,4.753,-44.320,-179.799,5.703,148.949
C05459=1192.992,4.503,-44.307,-179.801,5.702,148.949
C05460=1192.997,4.253,-44.292,-179.804,5.702,148.950
C05461=1193.003,4.004,-44.279,-179.806,5.702,148.951
C05462=1193.007,3.754,-44.264,-179.808,5.701,148.951
C05463=1193.012,3.504,-44.250,-179.811,5.701,148.952
C05464=1193.017,3.256,-44.237,-179.814,5.700,148.953
C05465=1193.023,2.986,-44.222,-179.816,5.700,148.953
C05466=1193.028,2.717,-44.207,-179.819,5.699,148.954
C05467=1193.034,2.448,-44.192,-179.822,5.699,148.955
C05468=1193.039,2.179,-44.176,-179.825,5.698,148.955
C05469=1193.045,1.929,-44.163,-179.826,5.698,148.956
C05470=1193.049,1.679,-44.149,-179.829,5.697,148.957
C05471=1193.054,1.430,-44.134,-179.832,5.697,148.957
C05472=1193.060,1.181,-44.120,-179.834,5.696,148.958
C05473=1193.065,0.931,-44.107,-179.837,5.696,148.959
C05474=1193.069,0.681,-44.093,-179.839,5.695,148.959
C05475=1193.075,0.432,-44.079,-179.842,5.694,148.960
C05476=1193.080,0.182,-44.065,-179.845,5.694,148.960
C05477=1193.085,-0.068,-44.051,-179.847,5.693,148.961
C05478=1193.090,-0.317,-44.038,-179.849,5.692,148.962
C05479=1193.095,-0.567,-44.024,-179.852,5.692,148.962
C05480=1193.100,-0.816,-44.009,-179.855,5.692,148.963
C05481=1193.106,-1.066,-43.996,-179.857,5.692,148.964
C05482=1193.110,-1.315,-43.983,-179.859,5.691,148.964
